// TIA Portal project "Magazyn_v1" (V16)
// Vorlageprojekt für das Buch mit Zielsystem S7-1200

(* hardware
DEVICE "S7-1200-Station_1"  S7-1200 Station
   slot 0: "Baugruppenträger_0"  Rack  V1.0
   slot 1: "PLC_1"  CPU 1211C DC/DC/DC  6ES7 211-1AE40-0XB0  V4.1
DEVICE "HMI_1"  TP900 Comfort SIPLUS
   slot 0: "HMI_1"  TP900 Comfort SIPLUS  6AG1 124-0JC01-4AX0  16.0.0.0
   slot 1: "HMI_RT_1"  TP900 Comfort SIPLUS  6AG1 124-0JC01-4AX0  16.0.0.0
   slot 5: "HMI_1.IE_CP_1"  PROFINET Interface  16.0.0.0
      slot 1: "PROFINET Interface_1"  PROFINET Interface
         slot 1: "Port_1"  Port
         slot 2: "Port_2"  Port
   slot 7: "HMI_1.MPI/DP_CP_1"  MPI/DP Interface  16.0.0.0
*)

// ===== PLC "PLC_1"  CPU 1211C DC/DC/DC =====

VAR_GLOBAL   // PLC tag table "Standard-Variablentabelle"
   "M30.1" AT %M30.1 : Bool;
   "M30.2" AT %M30.2 : Bool;
   "Tag_1" AT %I0.6 : Bool;
   "Tag_2" AT %I0.7 : Bool;
   "Tag_3" AT %Q0.5 : Bool;
   "Tag_4" AT %Q0.6 : Bool;
   "Tag_5" AT %Q0.7 : Bool;
   "box_full" AT %M30.3 : Bool;
   "M1_Conveyor_sec1_1" AT %M30.4 : Bool;
   "M2_Conveyor_sec1_1" AT %M30.5 : Bool;
   "Tag_6" AT %Q1.0 : Bool;
   "M1_Conveyor_sec1_2" AT %M30.6 : Bool;
   "M2_Conveyor_sec1_2" AT %M30.7 : Bool;
   "M1_Conveyor_sec1_3" AT %M31.0 : Bool;
   "M1_Conveyor_sec1_4" AT %M31.2 : Bool;
   "M2_Conveyor_sec1_4" AT %M31.3 : Bool;
   "M1_Conveyor_sec1_5" AT %M31.4 : Bool;
   "M2_Conveyor_sec1_5" AT %M31.5 : Bool;
   "M1_Conveyor_sec1_6" AT %M31.6 : Bool;
   "M2_Conveyor_sec1_6" AT %M31.7 : Bool;
   "M1_Conveyor_sec1_7" AT %M32.0 : Bool;
   "M2_Conveyor_sec1_7" AT %M32.1 : Bool;
   "Tag_7" AT %M32.2 : Bool;
   "pallet_fork_under_box_temp1" AT %M33.0 : Bool;
   "lift_box_temp1" AT %M33.1 : Bool;
   "ready_to_set_up_temp1" AT %M33.2 : Bool;
   "pallet_fork_storage_temp1" AT %M33.3 : Bool;
   "lower_box_temp1" AT %M33.4 : Bool;
   "pallet_fork_storage_withdraw_temp1" AT %M33.5 : Bool;
   "finish_stacker_Crane_sec1" AT %M33.6 : Bool;
   "Tag_8" AT %M33.7 : Bool;
   "is_pallete_elevator" AT %M34.0 : Bool;
   "_move_pallete_temp1" AT %M34.1 : Bool;
   "_move_pallete_temp2" AT %M34.2 : Bool;
   "_move_pallete_temp3" AT %M34.3 : Bool;
   "_move_pallete_temp4" AT %M34.5 : Bool;
   "set_is_pallere" AT %M34.6 : Bool;
   "Tag_9" AT %M34.4 : Bool;
   "pallete_ready_to_load" AT %M34.7 : Bool;
   "palletizing_box" AT %M35.0 : Bool;
   "pop_up_box_M" AT %M35.1 : Bool;
   "pop_up_palletizing_box" AT %M35.2 : Bool;
   "belt_conv_sec2_1_palletizing_box" AT %M35.3 : Bool;
   "belt_conv_sec2_1_palletizing_box_1" AT %M35.4 : Bool;
   "turn_box" AT %MW4 : Int;
   "belt_conv_sec2_1_palletizing_box_2" AT %M35.5 : Bool;
   "parallel_level" AT %M35.6 : Bool;
   "palletizer_finish_level" AT %M35.7 : Bool;
   "pallete_to_storage" AT %M36.0 : Bool;
   "palletizer_elevator_temp1" AT %M36.1 : Bool;
   "pallete_down_temp1" AT %M36.2 : Bool;
   "pallete_to_storage1" AT %M36.3 : Bool;
   "pallete_to_storage3" AT %M36.4 : Bool;
   "pallete_next_load" AT %M36.5 : Bool;
   "pallete_to_storage2" AT %M36.6 : Bool;
   "pallete_to_storage4" AT %M36.7 : Bool;
   "ready_to_set_up_temp1_2" AT %M37.0 : Bool;
   "pallet_fork_under_box_temp1_2" AT %M37.1 : Bool;
   "Tag_10" AT %M37.7 : Bool;
   "Tag_11" AT %M38.0 : Bool;
END_VAR

VAR_GLOBAL   // PLC tag table "Input_Variables_Factory"
   "FactoryIORunning" AT %I0.0 : Bool;
   "FactoryIOPaused" AT %I0.1 : Bool;
   "FactoryIOReset" AT %I0.2 : Bool;
   "Retroreflective Sensor 3 package" AT %I0.3 : Bool;
   "Retroreflective Sensor 4 Weight" AT %I0.4 : Bool;
   "Conveyor Scale 1 Weight (V)" AT %ID30 : Real;
   "M30.0" AT %M30.0 : Bool;
   "Retroreflective Sensor spad" AT %I0.5 : Bool;
   "Conveyor_sec1_1_Retroreflective Sensor" AT %I1.1 : Bool;
   "Conveyor_sec1_2_Retroreflective Sensor" AT %I1.2 : Bool;
   "Conveyor_sec1_3_Retroreflective Sensor" AT %I1.3 : Bool;
   "Conveyor_sec1_4_Retroreflective Sensor" AT %I1.4 : Bool;
   "Conveyor_sec1_5_Retroreflective Sensor" AT %I1.5 : Bool;
   "Conveyor_sec1_6_Retroreflective Sensor" AT %I1.6 : Bool;
   "Conveyor_sec1_7_storage_Retroreflective Sensor" AT %I1.7 : Bool;
   "M2_Conveyor_sec1_3" AT %M31.1 : Bool;
   "Roller_conveyor_sec2_down_1_Retroreflective_Sensor" AT %I2.0 : Bool;
   "Roller_conveyor_sec2_down_2_Retroreflective_Sensor" AT %I2.1 : Bool;
   "Belt_cinv_sec2_1_Retroreflective_Sensor" AT %I2.2 : Bool;
   "Palletizer 2 Elevator (Front Limit)" AT %I2.3 : Bool;
   "Loading_conv_sec2_Retroreflective_Sensor" AT %I2.4 : Bool;
   "Palletizer_Clamped_sensor" AT %I2.5 : Bool;
   "Palletizer_Plate_close" AT %I2.6 : Bool;
   "Palletizer_Pusher_Limit_sensor" AT %I2.7 : Bool;
   "Palletizer 2 Elevator (Back Limit)" AT %I1.0 : Bool;
   "lift_box_temp1_2" AT %M37.2 : Bool;
   "finish_stacker_Crane_sec1_2" AT %M37.3 : Bool;
   "pallet_fork_storage_temp1_2" AT %M37.4 : Bool;
   "lower_box_temp1_2" AT %M37.6 : Bool;
   "pallet_fork_storage_withdraw_temp1_2" AT %M37.5 : Bool;
   "Stacker Crane 2 Moving-X" AT %I3.0 : Bool;
   "Stacker Crane 2 Moving-Z" AT %I3.1 : Bool;
   "paletizer_counter" AT %MW6 : Int;
   "boxes_counter" AT %MW8 : Int;
   "paletizer_number_level" AT %MW16 : Int;
   "boxes_number_package" AT %MW18 : Int;
END_VAR

VAR_GLOBAL   // PLC tag table "Output_Variables_Factory"
   "Belt Conveyor (2m) 1 package" AT %Q0.0 : Bool;
   "Conveyor Scale 1 (+)" AT %Q0.1 : Bool;
   "Pop Up Wheel Sorter 2 (+)" AT %Q0.2 : Bool;
   "Pop Up Wheel Sorter 2 (Right)" AT %Q0.3 : Bool;
   "Belt Conveyor (2m) 7 przed spadem" AT %Q0.4 : Bool;
   "Conveyor_sec1_1" AT %Q1.1 : Bool;
   "Conveyor_sec1_2" AT %Q1.2 : Bool;
   "Conveyor_sec1_3" AT %Q1.3 : Bool;
   "Conveyor_sec1_4" AT %Q1.4 : Bool;
   "Conveyor_sec1_5" AT %Q1.5 : Bool;
   "Conveyor_sec1_6" AT %Q1.6 : Bool;
   "Conveyor_sec1_7_storage" AT %Q1.7 : Bool;
   "Stacker Crane sec1 under_box" AT %Q2.0 : Bool;
   "Stacker Crane sec1 Lift_box" AT %Q2.1 : Bool;
   "Stacker Crane sec1 storage" AT %Q2.2 : Bool;
   "Stacker Crane sec1 Target Position" AT %QD30 : DInt;
   "Belt_cinv_sec2_1" AT %Q2.3 : Bool;
   "Palletizer_belt_forward_sec_2_2" AT %Q2.4 : Bool;
   "Palletizer_turn" AT %Q2.5 : Bool;
   "Palletizer_push" AT %Q2.6 : Bool;
   "Palletizer_clamp" AT %Q2.7 : Bool;
   "Palletizer_open_plate" AT %Q3.0 : Bool;
   "Palletizer_elevator_limit" AT %Q3.1 : Bool;
   "Palletizer_elevator_up" AT %Q3.2 : Bool;
   "Palletizer_elevator_down" AT %Q3.3 : Bool;
   "Palletizer_chain_forward" AT %Q3.4 : Bool;
   "Roller_conveyor_sec2_down_1" AT %Q3.5 : Bool;
   "Roller_conveyor_sec2_down_2" AT %Q3.6 : Bool;
   "Loading_conv_sec2" AT %Q3.7 : Bool;
   "Stacker Crane 2 under_box" AT %Q4.0 : Bool;
   "Stacker Crane 2 Lift_box" AT %Q4.1 : Bool;
   "Stacker Crane 2 storage" AT %Q4.2 : Bool;
   "Stacker Crane 2 Target Position" AT %QD34 : DInt;
END_VAR

VAR_GLOBAL   // PLC tag table "Markers_outputs"
   "_Belt Conveyor (2m) 1 package" AT %M10.0 : Bool;
   "_Conveyor Scale 1 (+)" AT %M10.1 : Bool;
   "_Pop Up Wheel Sorter 2 (+)" AT %M10.2 : Bool;
   "_Pop Up Wheel Sorter 2 (Right)" AT %M10.3 : Bool;
   "_Belt Conveyor (2m) 7 przed spadem" AT %M10.4 : Bool;
   "M10.5" AT %M10.5 : Bool;
   "M10.6" AT %M10.6 : Bool;
   "M10.7" AT %M10.7 : Bool;
   "M11.0" AT %M11.0 : Bool;
   "_Conveyor_sec1_1" AT %M11.1 : Bool;
   "_Conveyor_sec1_2" AT %M11.2 : Bool;
   "_Conveyor_sec1_3" AT %M11.3 : Bool;
   "_Conveyor_sec1_4" AT %M11.4 : Bool;
   "_Conveyor_sec1_5" AT %M11.5 : Bool;
   "_Conveyor_sec1_6" AT %M11.6 : Bool;
   "_Conveyor_sec1_7_storage" AT %M11.7 : Bool;
   "_Stacker Crane sec1 under_box" AT %M12.0 : Bool;
   "_Stacker Crane sec1 Lift_box" AT %M12.1 : Bool;
   "_Stacker Crane sec1 storage" AT %M12.2 : Bool;
   "_Belt_cinv_sec2_1" AT %M12.3 : Bool;
   "_Palletizer_belt_forward_sec_2_2" AT %M12.4 : Bool;
   "_Palletizer_turn" AT %M12.5 : Bool;
   "_Palletizer_push" AT %M12.6 : Bool;
   "_Palletizer_clamp" AT %M12.7 : Bool;
   "_Palletizer_open_plate" AT %M13.0 : Bool;
   "_Palletizer_elevator_limit" AT %M13.1 : Bool;
   "_Palletizer_elevator_up" AT %M13.2 : Bool;
   "_Palletizer_elevator_down" AT %M13.3 : Bool;
   "_Palletizer_chain_forward" AT %M13.4 : Bool;
   "_Roller_conveyor_sec2_down_1" AT %M13.5 : Bool;
   "_Roller_conveyor_sec2_down_2" AT %M13.6 : Bool;
   "_Loading_conv_sec2" AT %M13.7 : Bool;
   "_Stacker Crane 2 under_box" AT %M14.0 : Bool;
   "_Stacker Crane 2 Lift_box" AT %M14.1 : Bool;
   "_Stacker Crane 2 storage" AT %M14.2 : Bool;
   "M14.3" AT %M14.3 : Bool;
   "_Stacker Crane sec1 Target Position" AT %MD20 : DInt;
   "_Stacker Crane sec1 Target Position_temp" AT %MD24 : DInt;
   "_Stacker Crane 2 Target Position" AT %MD38 : DInt;
   "_Stacker Crane 2 Target Position_temp" AT %MD42 : DInt;
END_VAR

VAR_GLOBAL   // PLC tag table "Markers_inputs"
   "_FactoryIORunning" AT %M0.0 : Bool;
   "_FactoryIOPaused" AT %M0.1 : Bool;
   "_FactoryIOReset" AT %M0.2 : Bool;
   "_Retroreflective Sensor 3 package" AT %M0.3 : Bool;
   "_Retroreflective Sensor 4 Weight" AT %M0.4 : Bool;
   "_Retroreflective Sensor spad" AT %M0.5 : Bool;
   "M0.6(1)" AT %M0.6 : Bool;
   "M0.7(1)" AT %M0.7 : Bool;
   "_Palletizer 2 Elevator (Back Limit)" AT %M1.0 : Bool;
   "_Conveyor_sec1_1_Retroreflective Sensor" AT %M1.1 : Bool;
   "_Conveyor_sec1_2_Retroreflective Sensor" AT %M1.2 : Bool;
   "_Conveyor_sec1_3_Retroreflective Sensor" AT %M1.3 : Bool;
   "_Conveyor_sec1_4_Retroreflective Sensor" AT %M1.4 : Bool;
   "_Conveyor_sec1_5_Retroreflective Sensor" AT %M1.5 : Bool;
   "_Conveyor_sec1_6_Retroreflective Sensor" AT %M1.6 : Bool;
   "_Conveyor_sec1_7_storage_Retroreflective Sensor" AT %M1.7 : Bool;
   "_Roller_conveyor_sec2_down_1_Retroreflective_Sensor" AT %M2.0 : Bool;
   "_Roller_conveyor_sec2_down_2_Retroreflective_Sensor" AT %M2.1 : Bool;
   "_Belt_cinv_sec2_1_Retroreflective_Sensor" AT %M2.2 : Bool;
   "_Palletizer 2 Elevator (Front Limit)" AT %M2.3 : Bool;
   "_Loading_conv_sec2_Retroreflective_Sensor" AT %M2.4 : Bool;
   "_Palletizer_Clamped_sensor" AT %M2.5 : Bool;
   "_Palletizer_Plate_close" AT %M2.6 : Bool;
   "_Palletizer_Pusher_Limit_sensor" AT %M2.7 : Bool;
   "_Stacker Crane 2 Moving-X" AT %M3.0 : Bool;
   "_Stacker Crane 2 Moving-Z" AT %M3.1 : Bool;
   "M3.2(1)" AT %M3.2 : Bool;
   "M3.3(1)" AT %M3.3 : Bool;
   "M3.4(1)" AT %M3.4 : Bool;
   "M3.5(1)" AT %M3.5 : Bool;
END_VAR

// folder: System blocks/Program resources

DATA_BLOCK "IEC_Timer_0_DB"   // DB1
{ S7_Optimized_Access := 'TRUE' }
AUTHOR : Simatic
FAMILY : IEC
NAME : IEC_TMR
VERSION : 1.0
// stored: InstanceOfName IEC_TIMER
"IEC_TIMER"
BEGIN
END_DATA_BLOCK

DATA_BLOCK "IEC_Counter_0_DB"   // DB2
{ S7_Optimized_Access := 'TRUE' }
AUTHOR : Simatic
FAMILY : IEC
NAME : CNTR
VERSION : 1.0
// stored: InstanceOfName IEC_COUNTER
"IEC_COUNTER"
BEGIN
END_DATA_BLOCK

DATA_BLOCK "licznik_sekcja_I"   // DB3
{ S7_Optimized_Access := 'TRUE' }
AUTHOR : Simatic
FAMILY : IEC
NAME : CNTR
VERSION : 1.0
// stored: InstanceOfName IEC_COUNTER
"IEC_COUNTER"
BEGIN
END_DATA_BLOCK

DATA_BLOCK "delay_switch_off"   // DB4
{ S7_Optimized_Access := 'TRUE' }
AUTHOR : Simatic
FAMILY : IEC
NAME : IEC_TMR
VERSION : 1.0
// stored: InstanceOfName IEC_TIMER
"IEC_TIMER"
BEGIN
END_DATA_BLOCK

DATA_BLOCK "IEC_Timer_0_DB_1"   // DB5
{ S7_Optimized_Access := 'TRUE' }
AUTHOR : Simatic
FAMILY : IEC
NAME : IEC_TMR
VERSION : 1.0
// stored: InstanceOfName IEC_TIMER
"IEC_TIMER"
BEGIN
END_DATA_BLOCK

DATA_BLOCK "IEC_Timer_0_DB_2"   // DB6
{ S7_Optimized_Access := 'TRUE' }
AUTHOR : Simatic
FAMILY : IEC
NAME : IEC_TMR
VERSION : 1.0
// stored: InstanceOfName IEC_TIMER
"IEC_TIMER"
BEGIN
END_DATA_BLOCK

DATA_BLOCK "IEC_Timer_0_DB_3"   // DB7
{ S7_Optimized_Access := 'TRUE' }
AUTHOR : Simatic
FAMILY : IEC
NAME : IEC_TMR
VERSION : 1.0
// stored: InstanceOfName IEC_TIMER
"IEC_TIMER"
BEGIN
END_DATA_BLOCK

DATA_BLOCK "IEC_Timer_0_DB_4"   // DB8
{ S7_Optimized_Access := 'TRUE' }
AUTHOR : Simatic
FAMILY : IEC
NAME : IEC_TMR
VERSION : 1.0
// stored: InstanceOfName IEC_TIMER
"IEC_TIMER"
BEGIN
END_DATA_BLOCK

DATA_BLOCK "IEC_Timer_0_DB_5"   // DB9
{ S7_Optimized_Access := 'TRUE' }
AUTHOR : Simatic
FAMILY : IEC
NAME : IEC_TMR
VERSION : 1.0
// stored: InstanceOfName IEC_TIMER
"IEC_TIMER"
BEGIN
END_DATA_BLOCK

DATA_BLOCK "IEC_Timer_0_DB_6"   // DB10
{ S7_Optimized_Access := 'TRUE' }
AUTHOR : Simatic
FAMILY : IEC
NAME : IEC_TMR
VERSION : 1.0
// stored: InstanceOfName IEC_TIMER
"IEC_TIMER"
BEGIN
END_DATA_BLOCK

DATA_BLOCK "IEC_Timer_0_DB_7"   // DB11
{ S7_Optimized_Access := 'TRUE' }
AUTHOR : Simatic
FAMILY : IEC
NAME : IEC_TMR
VERSION : 1.0
// stored: InstanceOfName IEC_TIMER
"IEC_TIMER"
BEGIN
END_DATA_BLOCK

DATA_BLOCK "IEC_Timer_0_DB_13"   // DB12
{ S7_Optimized_Access := 'TRUE' }
AUTHOR : Simatic
FAMILY : IEC
NAME : IEC_TMR
VERSION : 1.0
// stored: InstanceOfName IEC_TIMER
"IEC_TIMER"
BEGIN
END_DATA_BLOCK

DATA_BLOCK "IEC_Counter_0_DB_3"   // DB13
{ S7_Optimized_Access := 'TRUE' }
AUTHOR : Simatic
FAMILY : IEC
NAME : CNTR
VERSION : 1.0
// stored: InstanceOfName IEC_COUNTER
"IEC_COUNTER"
BEGIN
END_DATA_BLOCK

DATA_BLOCK "IEC_Timer_0_DB_9"   // DB14
{ S7_Optimized_Access := 'TRUE' }
AUTHOR : Simatic
FAMILY : IEC
NAME : IEC_TMR
VERSION : 1.0
// stored: InstanceOfName IEC_TIMER
"IEC_TIMER"
BEGIN
END_DATA_BLOCK

DATA_BLOCK "IEC_Timer_0_DB_10"   // DB15
{ S7_Optimized_Access := 'TRUE' }
AUTHOR : Simatic
FAMILY : IEC
NAME : IEC_TMR
VERSION : 1.0
// stored: InstanceOfName IEC_TIMER
"IEC_TIMER"
BEGIN
END_DATA_BLOCK

DATA_BLOCK "IEC_Counter_0_DB_4"   // DB16
{ S7_Optimized_Access := 'TRUE' }
AUTHOR : Simatic
FAMILY : IEC
NAME : CNTR
VERSION : 1.0
// stored: InstanceOfName IEC_COUNTER
"IEC_COUNTER"
BEGIN
END_DATA_BLOCK

DATA_BLOCK "IEC_Timer_0_DB_14"   // DB18
{ S7_Optimized_Access := 'TRUE' }
AUTHOR : Simatic
FAMILY : IEC
NAME : IEC_TMR
VERSION : 1.0
// stored: InstanceOfName IEC_TIMER
"IEC_TIMER"
BEGIN
END_DATA_BLOCK

DATA_BLOCK "IEC_Timer_0_DB_15"   // DB19
{ S7_Optimized_Access := 'TRUE' }
AUTHOR : Simatic
FAMILY : IEC
NAME : IEC_TMR
VERSION : 1.0
// stored: InstanceOfName IEC_TIMER
"IEC_TIMER"
BEGIN
END_DATA_BLOCK

DATA_BLOCK "IEC_Timer_0_DB_16"   // DB20
{ S7_Optimized_Access := 'TRUE' }
AUTHOR : Simatic
FAMILY : IEC
NAME : IEC_TMR
VERSION : 1.0
// stored: InstanceOfName IEC_TIMER
"IEC_TIMER"
BEGIN
END_DATA_BLOCK

DATA_BLOCK "IEC_Timer_0_DB_17"   // DB21
{ S7_Optimized_Access := 'TRUE' }
AUTHOR : Simatic
FAMILY : IEC
NAME : IEC_TMR
VERSION : 1.0
// stored: InstanceOfName IEC_TIMER
"IEC_TIMER"
BEGIN
END_DATA_BLOCK

DATA_BLOCK "licznik_sekcja_II"   // DB22
{ S7_Optimized_Access := 'TRUE' }
AUTHOR : Simatic
FAMILY : IEC
NAME : CNTR
VERSION : 1.0
// stored: InstanceOfName IEC_COUNTER
"IEC_COUNTER"
BEGIN
END_DATA_BLOCK

DATA_BLOCK "IEC_Timer_0_DB_19"   // DB23
{ S7_Optimized_Access := 'TRUE' }
AUTHOR : Simatic
FAMILY : IEC
NAME : IEC_TMR
VERSION : 1.0
// stored: InstanceOfName IEC_TIMER
"IEC_TIMER"
BEGIN
END_DATA_BLOCK

DATA_BLOCK "licznik_sekcja_II_two_levels"   // DB24
{ S7_Optimized_Access := 'TRUE' }
AUTHOR : Simatic
FAMILY : IEC
NAME : CNTR
VERSION : 1.0
// stored: InstanceOfName IEC_COUNTER
"IEC_COUNTER"
BEGIN
END_DATA_BLOCK

DATA_BLOCK "IEC_Timer_0_DB_20"   // DB25
{ S7_Optimized_Access := 'TRUE' }
AUTHOR : Simatic
FAMILY : IEC
NAME : IEC_TMR
VERSION : 1.0
// stored: InstanceOfName IEC_TIMER
"IEC_TIMER"
BEGIN
END_DATA_BLOCK

DATA_BLOCK "IEC_Timer_0_DB_18"   // DB26
{ S7_Optimized_Access := 'TRUE' }
AUTHOR : Simatic
FAMILY : IEC
NAME : IEC_TMR
VERSION : 1.0
// stored: InstanceOfName IEC_TIMER
"IEC_TIMER"
BEGIN
END_DATA_BLOCK

DATA_BLOCK "IEC_Timer_0_DB_21"   // DB27
{ S7_Optimized_Access := 'TRUE' }
AUTHOR : Simatic
FAMILY : IEC
NAME : IEC_TMR
VERSION : 1.0
// stored: InstanceOfName IEC_TIMER
"IEC_TIMER"
BEGIN
END_DATA_BLOCK

DATA_BLOCK "IEC_Counter_0_DB_1"   // DB28
{ S7_Optimized_Access := 'TRUE' }
AUTHOR : Simatic
FAMILY : IEC
NAME : CNTR
VERSION : 1.0
// stored: InstanceOfName IEC_COUNTER
"IEC_COUNTER"
BEGIN
END_DATA_BLOCK

DATA_BLOCK "IEC_Timer_0_DB_22"   // DB29
{ S7_Optimized_Access := 'TRUE' }
AUTHOR : Simatic
FAMILY : IEC
NAME : IEC_TMR
VERSION : 1.0
// stored: InstanceOfName IEC_TIMER
"IEC_TIMER"
BEGIN
END_DATA_BLOCK

DATA_BLOCK "IEC_Timer_0_DB_23"   // DB30
{ S7_Optimized_Access := 'TRUE' }
AUTHOR : Simatic
FAMILY : IEC
NAME : IEC_TMR
VERSION : 1.0
// stored: InstanceOfName IEC_TIMER
"IEC_TIMER"
BEGIN
END_DATA_BLOCK

DATA_BLOCK "IEC_Timer_0_DB_24"   // DB31
{ S7_Optimized_Access := 'TRUE' }
AUTHOR : Simatic
FAMILY : IEC
NAME : IEC_TMR
VERSION : 1.0
// stored: InstanceOfName IEC_TIMER
"IEC_TIMER"
BEGIN
END_DATA_BLOCK

DATA_BLOCK "IEC_Timer_0_DB_25"   // DB32
{ S7_Optimized_Access := 'TRUE' }
AUTHOR : Simatic
FAMILY : IEC
NAME : IEC_TMR
VERSION : 1.0
// stored: InstanceOfName IEC_TIMER
"IEC_TIMER"
BEGIN
END_DATA_BLOCK

DATA_BLOCK "IEC_Counter_0_DB_2"   // DB33
{ S7_Optimized_Access := 'TRUE' }
AUTHOR : Simatic
FAMILY : IEC
NAME : CNTR
VERSION : 1.0
// stored: InstanceOfName IEC_COUNTER
"IEC_COUNTER"
BEGIN
END_DATA_BLOCK

DATA_BLOCK "IEC_Timer_0_DB_26"   // DB34
{ S7_Optimized_Access := 'TRUE' }
AUTHOR : Simatic
FAMILY : IEC
NAME : IEC_TMR
VERSION : 1.0
// stored: InstanceOfName IEC_TIMER
"IEC_TIMER"
BEGIN
END_DATA_BLOCK

DATA_BLOCK "IEC_Timer_0_DB_27"   // DB35
{ S7_Optimized_Access := 'TRUE' }
AUTHOR : Simatic
FAMILY : IEC
NAME : IEC_TMR
VERSION : 1.0
// stored: InstanceOfName IEC_TIMER
"IEC_TIMER"
BEGIN
END_DATA_BLOCK

DATA_BLOCK "IEC_Timer_0_DB_28"   // DB36
{ S7_Optimized_Access := 'TRUE' }
AUTHOR : Simatic
FAMILY : IEC
NAME : IEC_TMR
VERSION : 1.0
// stored: InstanceOfName IEC_TIMER
"IEC_TIMER"
BEGIN
END_DATA_BLOCK

DATA_BLOCK "IEC_Timer_0_DB_29"   // DB37
{ S7_Optimized_Access := 'TRUE' }
AUTHOR : Simatic
FAMILY : IEC
NAME : IEC_TMR
VERSION : 1.0
// stored: InstanceOfName IEC_TIMER
"IEC_TIMER"
BEGIN
END_DATA_BLOCK

DATA_BLOCK "IEC_Timer_0_DB_30"   // DB38
{ S7_Optimized_Access := 'TRUE' }
AUTHOR : Simatic
FAMILY : IEC
NAME : IEC_TMR
VERSION : 1.0
// stored: InstanceOfName IEC_TIMER
"IEC_TIMER"
BEGIN
END_DATA_BLOCK

DATA_BLOCK "IEC_Timer_0_DB_31"   // DB39
{ S7_Optimized_Access := 'TRUE' }
AUTHOR : Simatic
FAMILY : IEC
NAME : IEC_TMR
VERSION : 1.0
// stored: InstanceOfName IEC_TIMER
"IEC_TIMER"
BEGIN
END_DATA_BLOCK

DATA_BLOCK "IEC_Timer_0_DB_32"   // DB40
{ S7_Optimized_Access := 'TRUE' }
AUTHOR : Simatic
FAMILY : IEC
NAME : IEC_TMR
VERSION : 1.0
// stored: InstanceOfName IEC_TIMER
"IEC_TIMER"
BEGIN
END_DATA_BLOCK

DATA_BLOCK "IEC_Timer_0_DB_33"   // DB41
{ S7_Optimized_Access := 'TRUE' }
AUTHOR : Simatic
FAMILY : IEC
NAME : IEC_TMR
VERSION : 1.0
// stored: InstanceOfName IEC_TIMER
"IEC_TIMER"
BEGIN
END_DATA_BLOCK

DATA_BLOCK "IEC_Timer_0_DB_34"   // DB42
{ S7_Optimized_Access := 'TRUE' }
AUTHOR : Simatic
FAMILY : IEC
NAME : IEC_TMR
VERSION : 1.0
// stored: InstanceOfName IEC_TIMER
"IEC_TIMER"
BEGIN
END_DATA_BLOCK

DATA_BLOCK "IEC_Timer_0_DB_35"   // DB43
{ S7_Optimized_Access := 'TRUE' }
AUTHOR : Simatic
FAMILY : IEC
NAME : IEC_TMR
VERSION : 1.0
// stored: InstanceOfName IEC_TIMER
"IEC_TIMER"
BEGIN
END_DATA_BLOCK

DATA_BLOCK "IEC_Timer_0_DB_36"   // DB44
{ S7_Optimized_Access := 'TRUE' }
AUTHOR : Simatic
FAMILY : IEC
NAME : IEC_TMR
VERSION : 1.0
// stored: InstanceOfName IEC_TIMER
"IEC_TIMER"
BEGIN
END_DATA_BLOCK

DATA_BLOCK "IEC_Timer_0_DB_37"   // DB45
{ S7_Optimized_Access := 'TRUE' }
AUTHOR : Simatic
FAMILY : IEC
NAME : IEC_TMR
VERSION : 1.0
// stored: InstanceOfName IEC_TIMER
"IEC_TIMER"
BEGIN
END_DATA_BLOCK

DATA_BLOCK "IEC_Timer_0_DB_38"   // DB46
{ S7_Optimized_Access := 'TRUE' }
AUTHOR : Simatic
FAMILY : IEC
NAME : IEC_TMR
VERSION : 1.0
// stored: InstanceOfName IEC_TIMER
"IEC_TIMER"
BEGIN
END_DATA_BLOCK

// folder: (top level)

FUNCTION "stacker_crane_2" : Void   // FC1, LAD
{ S7_Optimized_Access := 'TRUE' }
VERSION : 0.1
   VAR_TEMP
      mem5 : Bool;
      mem6 : Bool;
      mem7 : Bool;
   END_VAR
   VAR_TEMP   // added for the SCL form of the ladder/FBD networks
      _w1 : Bool;
      _w2 : Bool;
   END_VAR
BEGIN

REGION Network 2: Section1_pallete_fork
   // podjazd pod palete
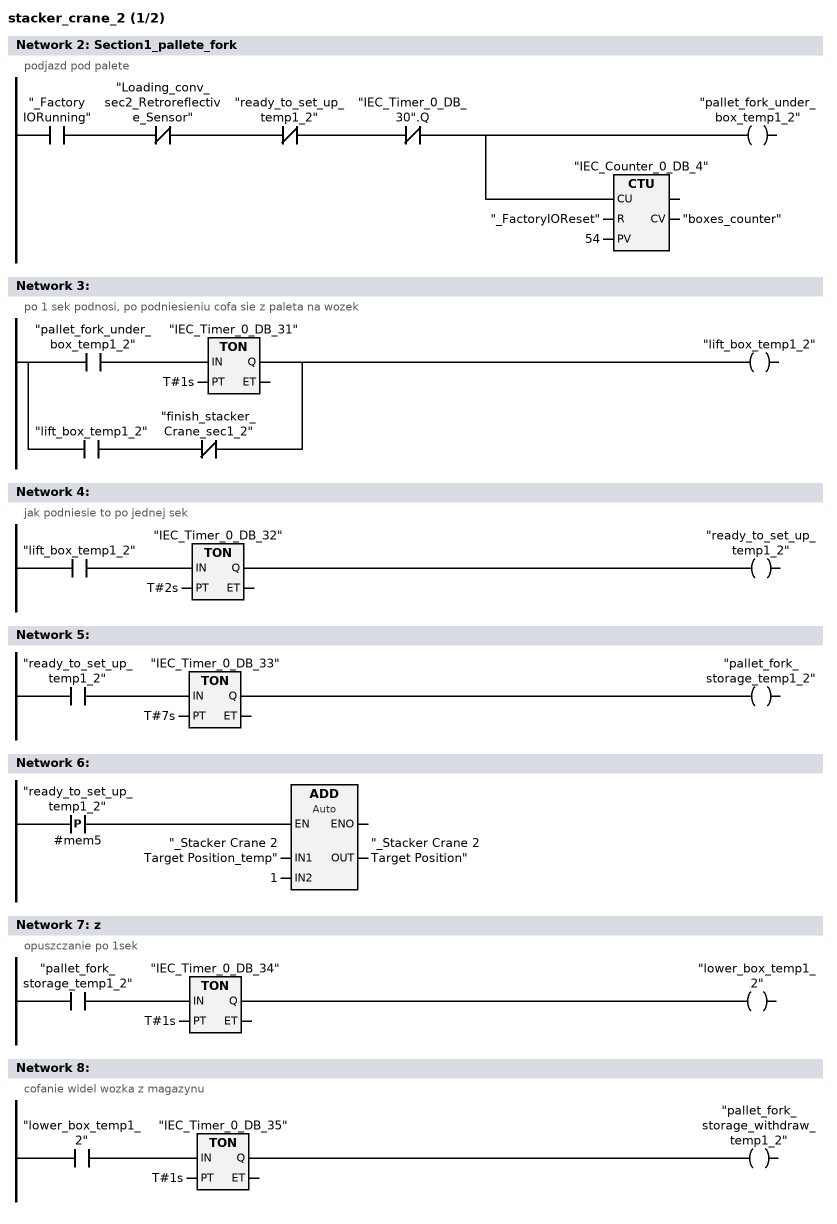
   "pallet_fork_under_box_temp1_2" := "_FactoryIORunning" AND NOT "Loading_conv_sec2_Retroreflective_Sensor" AND NOT "ready_to_set_up_temp1_2" AND NOT "IEC_Timer_0_DB_30".Q;
   "IEC_Counter_0_DB_4".CTU(CU := "pallet_fork_under_box_temp1_2",
                           R := "_FactoryIOReset",
                           PV := 54,
                           CV => "boxes_counter");
END_REGION

REGION Network 3
   // po 1 sek podnosi, po podniesieniu cofa sie z paleta na wozek
   "IEC_Timer_0_DB_31".TON(IN := "pallet_fork_under_box_temp1_2", PT := T#1s);
   "lift_box_temp1_2" := "IEC_Timer_0_DB_31".Q OR ("lift_box_temp1_2" AND NOT "finish_stacker_Crane_sec1_2");
END_REGION

REGION Network 4
   // jak podniesie to po jednej sek
   "IEC_Timer_0_DB_32".TON(IN := "lift_box_temp1_2", PT := T#2s);
   "ready_to_set_up_temp1_2" := "IEC_Timer_0_DB_32".Q;
END_REGION

REGION Network 5
   "IEC_Timer_0_DB_33".TON(IN := "ready_to_set_up_temp1_2", PT := T#7s);
   "pallet_fork_storage_temp1_2" := "IEC_Timer_0_DB_33".Q;
END_REGION

REGION Network 6
   RUNG wire#powerrail
      P_Contact(operand := "ready_to_set_up_temp1_2", bit := #mem5)
      Add(in1 := "_Stacker Crane 2 Target Position_temp", in2 := 1, out => "_Stacker Crane 2 Target Position")
   END_RUNG
   // the same network as SCL:
   #_w1 := "ready_to_set_up_temp1_2" AND NOT #mem5;   // rising edge of "ready_to_set_up_temp1_2"
   #mem5 := "ready_to_set_up_temp1_2";
   IF #_w1 THEN "_Stacker Crane 2 Target Position" := "_Stacker Crane 2 Target Position_temp" + 1; END_IF;
END_REGION

REGION Network 7: z
   // opuszczanie po 1sek
   "IEC_Timer_0_DB_34".TON(IN := "pallet_fork_storage_temp1_2", PT := T#1s);
   "lower_box_temp1_2" := "IEC_Timer_0_DB_34".Q;
END_REGION

REGION Network 8
   // cofanie widel wozka z magazynu
   "IEC_Timer_0_DB_35".TON(IN := "lower_box_temp1_2", PT := T#1s);
   "pallet_fork_storage_withdraw_temp1_2" := "IEC_Timer_0_DB_35".Q;
END_REGION

REGION Network 9
   // powrot na pozycje startowa widlaka
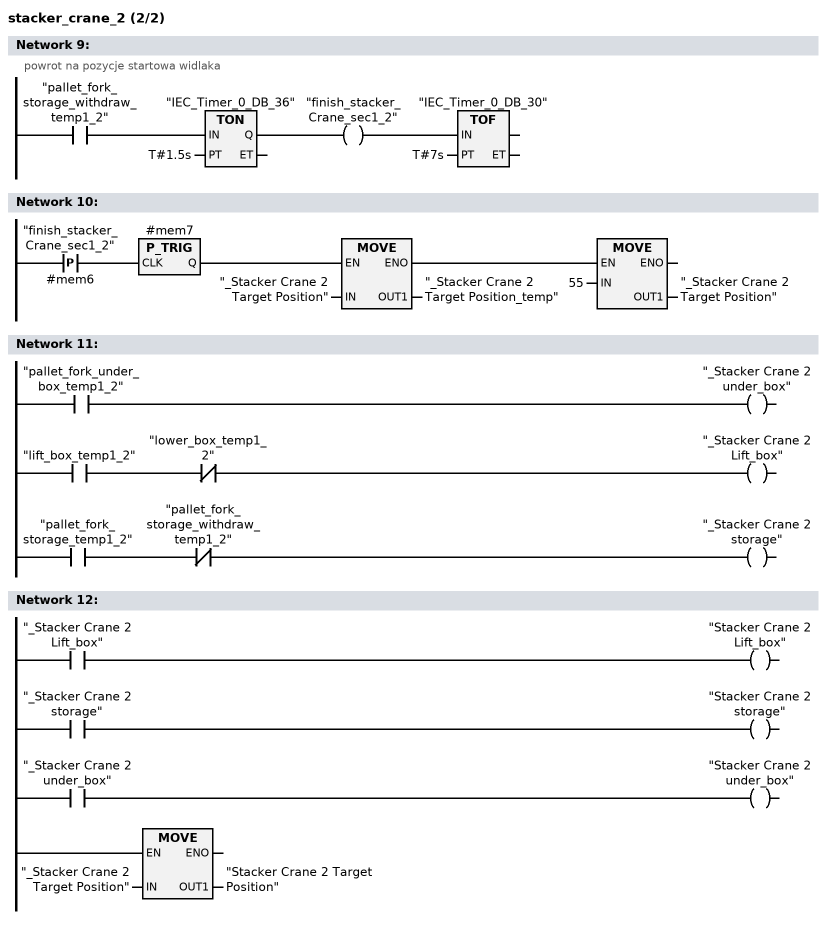
   "IEC_Timer_0_DB_36".TON(IN := "pallet_fork_storage_withdraw_temp1_2", PT := T#1.5s);
   "finish_stacker_Crane_sec1_2" := "IEC_Timer_0_DB_36".Q;
   "IEC_Timer_0_DB_30".TOF(IN := "IEC_Timer_0_DB_36".Q, PT := T#7s);
END_REGION

REGION Network 10
   RUNG wire#powerrail
      P_Contact(operand := "finish_stacker_Crane_sec1_2", bit := #mem6)
      P_Trig( #mem7 )
      Move(in := "_Stacker Crane 2 Target Position", out1 => "_Stacker Crane 2 Target Position_temp")
      Move(in := 55, out1 => "_Stacker Crane 2 Target Position")
   END_RUNG
   // the same network as SCL:
   #_w1 := "finish_stacker_Crane_sec1_2" AND NOT #mem6;   // rising edge of "finish_stacker_Crane_sec1_2"
   #mem6 := "finish_stacker_Crane_sec1_2";
   #_w2 := #_w1 AND NOT #mem7;   // rising edge
   #mem7 := #_w1;
   IF #_w2 THEN
       "_Stacker Crane 2 Target Position_temp" := "_Stacker Crane 2 Target Position";
       "_Stacker Crane 2 Target Position" := 55;
   END_IF;
END_REGION

REGION Network 11
   RUNG wire#powerrail
      Contact( "pallet_fork_under_box_temp1_2" )
      Coil( "_Stacker Crane 2 under_box" )
   END_RUNG
   RUNG wire#powerrail
      Contact( "lift_box_temp1_2" )
      I_Contact( "lower_box_temp1_2" )
      Coil( "_Stacker Crane 2 Lift_box" )
   END_RUNG
   RUNG wire#powerrail
      Contact( "pallet_fork_storage_temp1_2" )
      I_Contact( "pallet_fork_storage_withdraw_temp1_2" )
      Coil( "_Stacker Crane 2 storage" )
   END_RUNG
   // the same network as SCL:
   "_Stacker Crane 2 under_box" := "pallet_fork_under_box_temp1_2";
   "_Stacker Crane 2 Lift_box" := "lift_box_temp1_2" AND NOT "lower_box_temp1_2";
   "_Stacker Crane 2 storage" := "pallet_fork_storage_temp1_2" AND NOT "pallet_fork_storage_withdraw_temp1_2";
END_REGION

REGION Network 12
   RUNG wire#powerrail
      Contact( "_Stacker Crane 2 Lift_box" )
      Coil( "Stacker Crane 2 Lift_box" )
   END_RUNG
   RUNG wire#powerrail
      Contact( "_Stacker Crane 2 storage" )
      Coil( "Stacker Crane 2 storage" )
   END_RUNG
   RUNG wire#powerrail
      Contact( "_Stacker Crane 2 under_box" )
      Coil( "Stacker Crane 2 under_box" )
   END_RUNG
   RUNG wire#powerrail
      Move(in := "_Stacker Crane 2 Target Position", out1 => "Stacker Crane 2 Target Position")
   END_RUNG
   // the same network as SCL:
   "Stacker Crane 2 Lift_box" := "_Stacker Crane 2 Lift_box";
   "Stacker Crane 2 storage" := "_Stacker Crane 2 storage";
   "Stacker Crane 2 under_box" := "_Stacker Crane 2 under_box";
   "Stacker Crane 2 Target Position" := "_Stacker Crane 2 Target Position";
END_REGION
END_FUNCTION

FUNCTION "MHJ-PLC-Lab-Function-S71200" : Void   // FC9000, SCL
{ S7_Optimized_Access := 'TRUE' }
VERSION : 0.1
   VAR_TEMP
      rdTimeReturn : Int;
      outputTime : DTL;
      SyncVal : Byte;
      forVal : Int;
      forVal_2 : Int;
      Value : Byte;
   END_VAR
   VAR CONSTANT
      CompVal : Byte := 16#34;
      Value_01 : Byte := 16#11;
      Value_01_DW : DWord := 16#A165_D992;
      Value_02_DW : DWord := 16#58BE_4401;
   END_VAR
BEGIN

   #Value:=PEEK(area := 16#82,
        dbNumber := 0,
        byteOffset := 511);
   #Value := #Value + 1;

   POKE(area := 16#82,
        dbNumber := 0,
        byteOffset := 511,
        value := #Value);

   POKE(area:=16#81,
        dbNumber:=0,
        byteOffset:=1016,
        value:=#Value_01_DW);
   POKE(area := 16#81,
        dbNumber := 0,
        byteOffset := 1020,
        value := #Value_02_DW);

   POKE(area := 16#81,
        dbNumber := 0,
        byteOffset := 511,
        value := B#16#00);

   FOR #forVal := 0 TO 120 DO
       FOR #forVal_2:=0 TO 10 DO
           #rdTimeReturn:=RD_SYS_T(#outputTime);
           #rdTimeReturn := WR_SYS_T(#outputTime);
           #rdTimeReturn := RD_SYS_T(#outputTime);
           #rdTimeReturn := WR_SYS_T(#outputTime);
       END_FOR;
       #SyncVal:= PEEK(area := 16#81,
                      dbNumber := 0,
                      byteOffset := 511);
       IF #SyncVal = #CompVal THEN
          GOTO M_1;
       END_IF;
   END_FOR;
   RETURN;

   M_1:
   POKE(area := 16#81,
        dbNumber := 0,
        byteOffset := 511,
        value := B#16#0);
END_FUNCTION

ORGANIZATION_BLOCK "Main"   // OB1, LAD, ProgramCycle
TITLE = "Main Program Sweep (Cycle)"
{ S7_Optimized_Access := 'TRUE' }
VERSION : 0.1
   VAR_INPUT
      Initial_Call : Bool;   // Initial call of this OB
      Remanence : Bool;   // =True, if remanent data are available
   END_VAR
   VAR_TEMP
      mem1 : Bool;
      mem2 : Bool;
      mem3 : Bool;
      _box_full : Bool;
      M1_Conveyor_sec1_1 : Bool;
      M2_Conveyor_sec1_1 : Bool;
      mem4 : Bool;
      mem5 : Bool;
      mem6 : Bool;
      mem7 : Bool;
      mem8 : Bool;
      sr1 : Bool;
      sr2 : Bool;
      mem9 : Bool;
      mem10 : Bool;
      mem11 : Bool;
      mem12 : Bool;
      mem13 : Bool;
      mem14 : Bool;
      mem15 : Bool;
      mem16 : Bool;
      mem17 : Bool;
      mem18 : Bool;
      mem19 : Bool;
      mem20 : Bool;
   END_VAR
   VAR_TEMP   // added for the SCL form of the ladder/FBD networks
      _w1 : Bool;
      _w2 : Bool;
   END_VAR
BEGIN

REGION Network 1: Konnektierungsbaustein für PLC-Lab
   // Im Netzwerk 1 wird der Konnektierungsbaustein für PLC-Lab aufgerufen.
   // Dieser Aufruf darf nicht entfernt werden!
   // Enable connention with Factory I/O
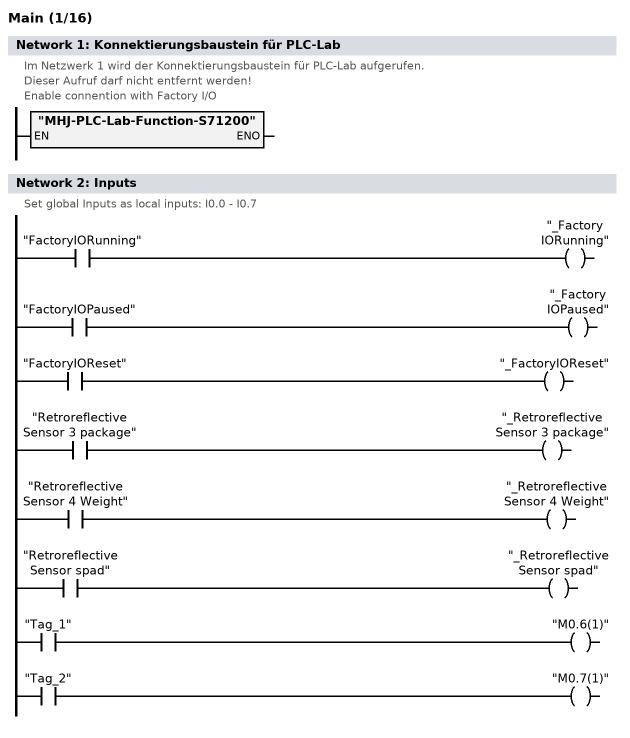
   RUNG wire#powerrail
      "MHJ-PLC-Lab-Function-S71200"()
   END_RUNG
   // the same network as SCL:
   "MHJ-PLC-Lab-Function-S71200"();
END_REGION

REGION Network 2: Inputs
   // Set global Inputs as local inputs: I0.0 - I0.7
   RUNG wire#powerrail
      Contact( "FactoryIORunning" )
      Coil( "_FactoryIORunning" )
   END_RUNG
   RUNG wire#powerrail
      Contact( "FactoryIOPaused" )
      Coil( "_FactoryIOPaused" )
   END_RUNG
   RUNG wire#powerrail
      Contact( "FactoryIOReset" )
      Coil( "_FactoryIOReset" )
   END_RUNG
   RUNG wire#powerrail
      Contact( "Retroreflective Sensor 3 package" )
      Coil( "_Retroreflective Sensor 3 package" )
   END_RUNG
   RUNG wire#powerrail
      Contact( "Retroreflective Sensor 4 Weight" )
      Coil( "_Retroreflective Sensor 4 Weight" )
   END_RUNG
   RUNG wire#powerrail
      Contact( "Retroreflective Sensor spad" )
      Coil( "_Retroreflective Sensor spad" )
   END_RUNG
   RUNG wire#powerrail
      Contact( "Tag_1" )
      Coil( "M0.6(1)" )
   END_RUNG
   RUNG wire#powerrail
      Contact( "Tag_2" )
      Coil( "M0.7(1)" )
   END_RUNG
   // the same network as SCL:
   "_FactoryIORunning" := "FactoryIORunning";
   "_FactoryIOPaused" := "FactoryIOPaused";
   "_FactoryIOReset" := "FactoryIOReset";
   "_Retroreflective Sensor 3 package" := "Retroreflective Sensor 3 package";
   "_Retroreflective Sensor 4 Weight" := "Retroreflective Sensor 4 Weight";
   "_Retroreflective Sensor spad" := "Retroreflective Sensor spad";
   "M0.6(1)" := "Tag_1";
   "M0.7(1)" := "Tag_2";
END_REGION

REGION Network 3
   // Set global Inputs as local inputs: I1.0 - I1.7
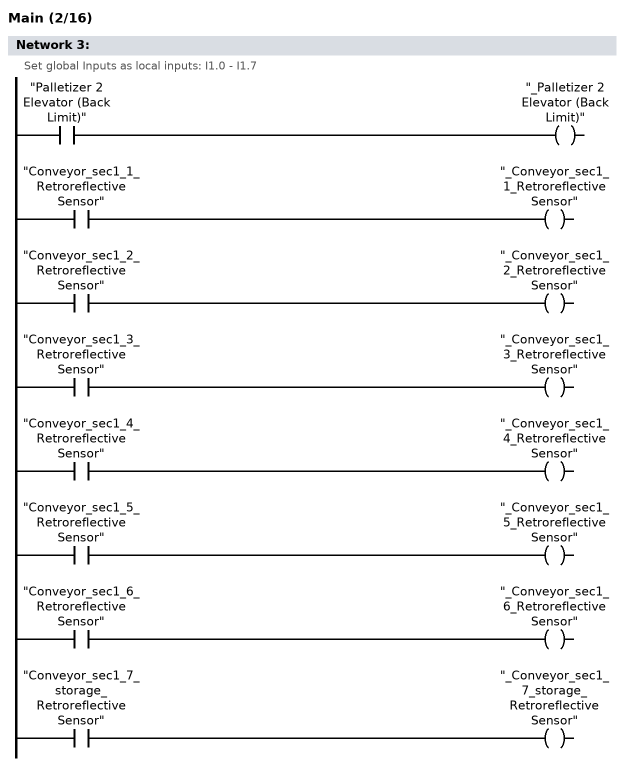
   RUNG wire#powerrail
      Contact( "Palletizer 2 Elevator (Back Limit)" )
      Coil( "_Palletizer 2 Elevator (Back Limit)" )
   END_RUNG
   RUNG wire#powerrail
      Contact( "Conveyor_sec1_1_Retroreflective Sensor" )
      Coil( "_Conveyor_sec1_1_Retroreflective Sensor" )
   END_RUNG
   RUNG wire#powerrail
      Contact( "Conveyor_sec1_2_Retroreflective Sensor" )
      Coil( "_Conveyor_sec1_2_Retroreflective Sensor" )
   END_RUNG
   RUNG wire#powerrail
      Contact( "Conveyor_sec1_3_Retroreflective Sensor" )
      Coil( "_Conveyor_sec1_3_Retroreflective Sensor" )
   END_RUNG
   RUNG wire#powerrail
      Contact( "Conveyor_sec1_4_Retroreflective Sensor" )
      Coil( "_Conveyor_sec1_4_Retroreflective Sensor" )
   END_RUNG
   RUNG wire#powerrail
      Contact( "Conveyor_sec1_5_Retroreflective Sensor" )
      Coil( "_Conveyor_sec1_5_Retroreflective Sensor" )
   END_RUNG
   RUNG wire#powerrail
      Contact( "Conveyor_sec1_6_Retroreflective Sensor" )
      Coil( "_Conveyor_sec1_6_Retroreflective Sensor" )
   END_RUNG
   RUNG wire#powerrail
      Contact( "Conveyor_sec1_7_storage_Retroreflective Sensor" )
      Coil( "_Conveyor_sec1_7_storage_Retroreflective Sensor" )
   END_RUNG
   // the same network as SCL:
   "_Palletizer 2 Elevator (Back Limit)" := "Palletizer 2 Elevator (Back Limit)";
   "_Conveyor_sec1_1_Retroreflective Sensor" := "Conveyor_sec1_1_Retroreflective Sensor";
   "_Conveyor_sec1_2_Retroreflective Sensor" := "Conveyor_sec1_2_Retroreflective Sensor";
   "_Conveyor_sec1_3_Retroreflective Sensor" := "Conveyor_sec1_3_Retroreflective Sensor";
   "_Conveyor_sec1_4_Retroreflective Sensor" := "Conveyor_sec1_4_Retroreflective Sensor";
   "_Conveyor_sec1_5_Retroreflective Sensor" := "Conveyor_sec1_5_Retroreflective Sensor";
   "_Conveyor_sec1_6_Retroreflective Sensor" := "Conveyor_sec1_6_Retroreflective Sensor";
   "_Conveyor_sec1_7_storage_Retroreflective Sensor" := "Conveyor_sec1_7_storage_Retroreflective Sensor";
END_REGION

REGION Network 4
   // Set global Inputs as local inputs: I2.0 - I2.7
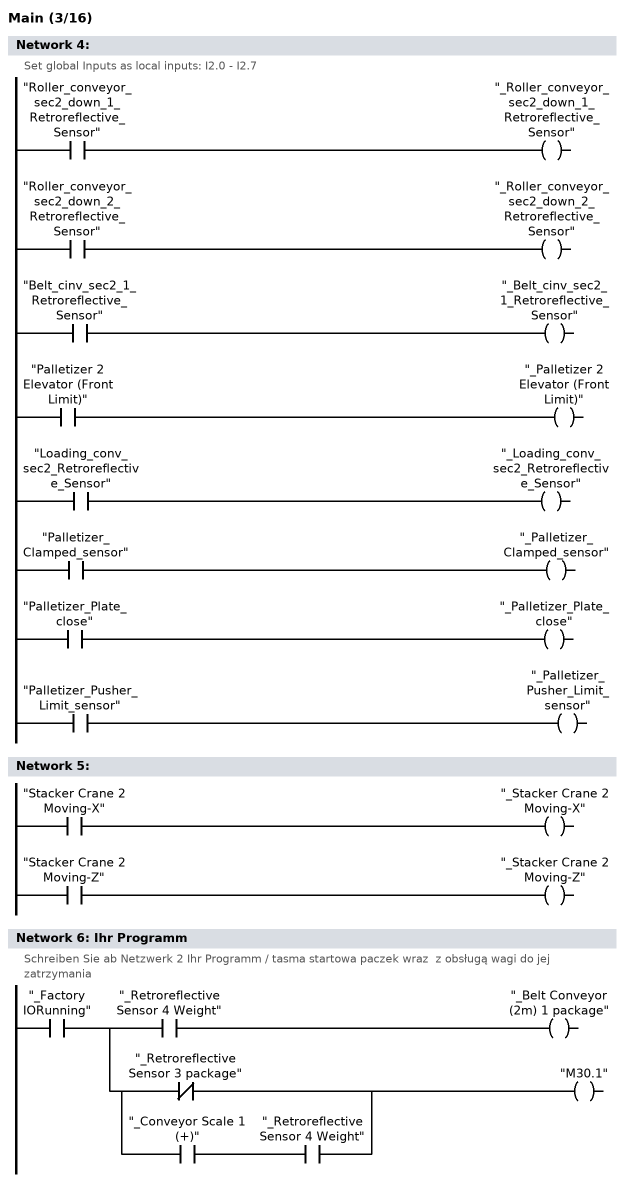
   RUNG wire#powerrail
      Contact( "Roller_conveyor_sec2_down_1_Retroreflective_Sensor" )
      Coil( "_Roller_conveyor_sec2_down_1_Retroreflective_Sensor" )
   END_RUNG
   RUNG wire#powerrail
      Contact( "Roller_conveyor_sec2_down_2_Retroreflective_Sensor" )
      Coil( "_Roller_conveyor_sec2_down_2_Retroreflective_Sensor" )
   END_RUNG
   RUNG wire#powerrail
      Contact( "Belt_cinv_sec2_1_Retroreflective_Sensor" )
      Coil( "_Belt_cinv_sec2_1_Retroreflective_Sensor" )
   END_RUNG
   RUNG wire#powerrail
      Contact( "Palletizer 2 Elevator (Front Limit)" )
      Coil( "_Palletizer 2 Elevator (Front Limit)" )
   END_RUNG
   RUNG wire#powerrail
      Contact( "Loading_conv_sec2_Retroreflective_Sensor" )
      Coil( "_Loading_conv_sec2_Retroreflective_Sensor" )
   END_RUNG
   RUNG wire#powerrail
      Contact( "Palletizer_Clamped_sensor" )
      Coil( "_Palletizer_Clamped_sensor" )
   END_RUNG
   RUNG wire#powerrail
      Contact( "Palletizer_Plate_close" )
      Coil( "_Palletizer_Plate_close" )
   END_RUNG
   RUNG wire#powerrail
      Contact( "Palletizer_Pusher_Limit_sensor" )
      Coil( "_Palletizer_Pusher_Limit_sensor" )
   END_RUNG
   // the same network as SCL:
   "_Roller_conveyor_sec2_down_1_Retroreflective_Sensor" := "Roller_conveyor_sec2_down_1_Retroreflective_Sensor";
   "_Roller_conveyor_sec2_down_2_Retroreflective_Sensor" := "Roller_conveyor_sec2_down_2_Retroreflective_Sensor";
   "_Belt_cinv_sec2_1_Retroreflective_Sensor" := "Belt_cinv_sec2_1_Retroreflective_Sensor";
   "_Palletizer 2 Elevator (Front Limit)" := "Palletizer 2 Elevator (Front Limit)";
   "_Loading_conv_sec2_Retroreflective_Sensor" := "Loading_conv_sec2_Retroreflective_Sensor";
   "_Palletizer_Clamped_sensor" := "Palletizer_Clamped_sensor";
   "_Palletizer_Plate_close" := "Palletizer_Plate_close";
   "_Palletizer_Pusher_Limit_sensor" := "Palletizer_Pusher_Limit_sensor";
END_REGION

REGION Network 5
   RUNG wire#powerrail
      Contact( "Stacker Crane 2 Moving-X" )
      Coil( "_Stacker Crane 2 Moving-X" )
   END_RUNG
   RUNG wire#powerrail
      Contact( "Stacker Crane 2 Moving-Z" )
      Coil( "_Stacker Crane 2 Moving-Z" )
   END_RUNG
   // the same network as SCL:
   "_Stacker Crane 2 Moving-X" := "Stacker Crane 2 Moving-X";
   "_Stacker Crane 2 Moving-Z" := "Stacker Crane 2 Moving-Z";
END_REGION

REGION Network 6: Ihr Programm
   // Schreiben Sie ab Netzwerk 2 Ihr Programm / tasma startowa paczek wraz  z obsługą wagi do jej zatrzymania
   RUNG wire#powerrail
      Contact( "_FactoryIORunning" )
      wire#w1
      Contact( "_Retroreflective Sensor 4 Weight" )
      Coil( "_Belt Conveyor (2m) 1 package" )
   END_RUNG
   RUNG wire#w1
      I_Contact( "_Retroreflective Sensor 3 package" )
      wire#w2
      Coil( "M30.1" )
   END_RUNG
   RUNG wire#w1
      Contact( "_Conveyor Scale 1 (+)" )
      Contact( "_Retroreflective Sensor 4 Weight" )
   END_RUNG wire#w2
   // the same network as SCL:
   "_Belt Conveyor (2m) 1 package" := "_FactoryIORunning" AND "_Retroreflective Sensor 4 Weight";
   "M30.1" := "_FactoryIORunning" AND (NOT "_Retroreflective Sensor 3 package" OR ("_Conveyor Scale 1 (+)" AND "_Retroreflective Sensor 4 Weight"));
END_REGION

REGION Network 7
   // rolki dla paczki M oraz zalaczenie tasmy - warunki
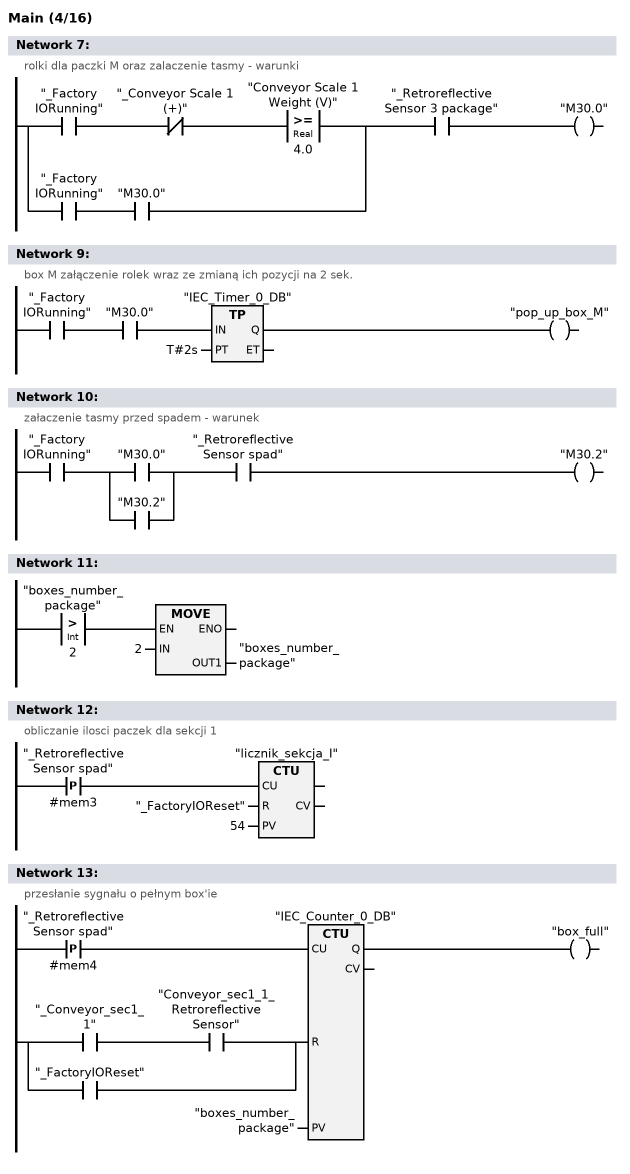
   RUNG wire#powerrail
      Contact( "_FactoryIORunning" )
      I_Contact( "_Conveyor Scale 1 (+)" )
      { S7_Templates := "SrcType := Real" } GE_Contact(in1 := "Conveyor Scale 1 Weight (V)", in2 := 4.0)
      wire#w1
      Contact( "_Retroreflective Sensor 3 package" )
      Coil( "M30.0" )
   END_RUNG
   RUNG wire#powerrail
      Contact( "_FactoryIORunning" )
      Contact( "M30.0" )
   END_RUNG wire#w1
   // the same network as SCL:
   "M30.0" := (("_FactoryIORunning" AND NOT "_Conveyor Scale 1 (+)" AND ("Conveyor Scale 1 Weight (V)" >= 4.0)) OR ("_FactoryIORunning" AND "M30.0")) AND "_Retroreflective Sensor 3 package";
END_REGION

REGION Network 9
   // box M załączenie rolek wraz ze zmianą ich pozycji na 2 sek.
   "IEC_Timer_0_DB".TP(IN := "_FactoryIORunning" AND "M30.0", PT := T#2s);
   "pop_up_box_M" := "IEC_Timer_0_DB".Q;
END_REGION

REGION Network 10
   // załaczenie tasmy przed spadem - warunek
   RUNG wire#powerrail
      Contact( "_FactoryIORunning" )
      wire#w1
      Contact( "M30.0" )
      wire#w2
      Contact( "_Retroreflective Sensor spad" )
      Coil( "M30.2" )
   END_RUNG
   RUNG wire#w1
      Contact( "M30.2" )
   END_RUNG wire#w2
   // the same network as SCL:
   "M30.2" := "_FactoryIORunning" AND ("M30.0" OR "M30.2") AND "_Retroreflective Sensor spad";
END_REGION

REGION Network 11
   RUNG wire#powerrail
      { S7_Templates := "SrcType := Int" } GT_Contact(in1 := "boxes_number_package", in2 := 2)
      Move(in := 2, out1 => "boxes_number_package")
   END_RUNG
   // the same network as SCL:
   IF "boxes_number_package" > 2 THEN "boxes_number_package" := 2; END_IF;
END_REGION

REGION Network 12
   // obliczanie ilosci paczek dla sekcji 1
   #_w1 := "_Retroreflective Sensor spad" AND NOT #mem3;   // rising edge of "_Retroreflective Sensor spad"
   #mem3 := "_Retroreflective Sensor spad";
   "licznik_sekcja_I".CTU(CU := #_w1, R := "_FactoryIOReset", PV := 54);
END_REGION

REGION Network 13
   // przesłanie sygnału o pełnym box'ie
   #_w1 := "_Retroreflective Sensor spad" AND NOT #mem4;   // rising edge of "_Retroreflective Sensor spad"
   #mem4 := "_Retroreflective Sensor spad";
   "IEC_Counter_0_DB".CTU(CU := #_w1,
                          R := ("_Conveyor_sec1_1" AND "Conveyor_sec1_1_Retroreflective Sensor") OR "_FactoryIOReset",
                          PV := "boxes_number_package");
   "box_full" := "IEC_Counter_0_DB".Q;
END_REGION

REGION Network 14
   // zalaczenie tasmy,aby box dojechal po odbior paczki
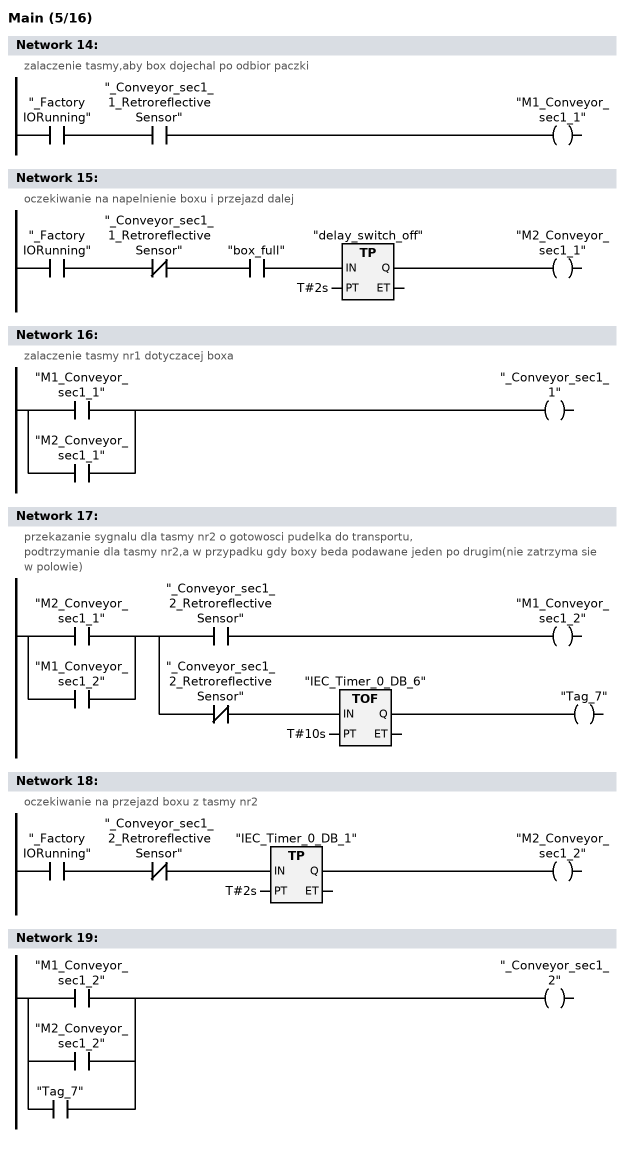
   RUNG wire#powerrail
      Contact( "_FactoryIORunning" )
      Contact( "_Conveyor_sec1_1_Retroreflective Sensor" )
      Coil( "M1_Conveyor_sec1_1" )
   END_RUNG
   // the same network as SCL:
   "M1_Conveyor_sec1_1" := "_FactoryIORunning" AND "_Conveyor_sec1_1_Retroreflective Sensor";
END_REGION

REGION Network 15
   // oczekiwanie na napelnienie boxu i przejazd dalej
   "delay_switch_off".TP(IN := "_FactoryIORunning" AND NOT "_Conveyor_sec1_1_Retroreflective Sensor" AND "box_full",
                         PT := T#2s);
   "M2_Conveyor_sec1_1" := "delay_switch_off".Q;
END_REGION

REGION Network 16
   // zalaczenie tasmy nr1 dotyczacej boxa
   RUNG wire#powerrail
      Contact( "M1_Conveyor_sec1_1" )
      wire#w1
      Coil( "_Conveyor_sec1_1" )
   END_RUNG
   RUNG wire#powerrail
      Contact( "M2_Conveyor_sec1_1" )
   END_RUNG wire#w1
   // the same network as SCL:
   "_Conveyor_sec1_1" := "M1_Conveyor_sec1_1" OR "M2_Conveyor_sec1_1";
END_REGION

REGION Network 17
   // przekazanie sygnalu dla tasmy nr2 o gotowosci pudelka do transportu, 
   // podtrzymanie dla tasmy nr2,a w przypadku gdy boxy beda podawane jeden po drugim(nie zatrzyma sie w polowie)
   #_w1 := "M2_Conveyor_sec1_1" OR "M1_Conveyor_sec1_2";
   "M1_Conveyor_sec1_2" := #_w1 AND "_Conveyor_sec1_2_Retroreflective Sensor";
   "IEC_Timer_0_DB_6".TOF(IN := #_w1 AND NOT "_Conveyor_sec1_2_Retroreflective Sensor", PT := T#10s);
   "Tag_7" := "IEC_Timer_0_DB_6".Q;
END_REGION

REGION Network 18
   // oczekiwanie na przejazd boxu z tasmy nr2
   "IEC_Timer_0_DB_1".TP(IN := "_FactoryIORunning" AND NOT "_Conveyor_sec1_2_Retroreflective Sensor",
                         PT := T#2s);
   "M2_Conveyor_sec1_2" := "IEC_Timer_0_DB_1".Q;
END_REGION

REGION Network 19
   RUNG wire#powerrail
      Contact( "M1_Conveyor_sec1_2" )
      wire#w1
      Coil( "_Conveyor_sec1_2" )
   END_RUNG
   RUNG wire#powerrail
      Contact( "M2_Conveyor_sec1_2" )
   END_RUNG wire#w1
   RUNG wire#powerrail
      Contact( "Tag_7" )
   END_RUNG wire#w1
   // the same network as SCL:
   "_Conveyor_sec1_2" := "M1_Conveyor_sec1_2" OR "M2_Conveyor_sec1_2" OR "Tag_7";
END_REGION

REGION Network 20
   // przekazanie sygnalu dla tasmy nr3 o gotowosci pudelka do transportu
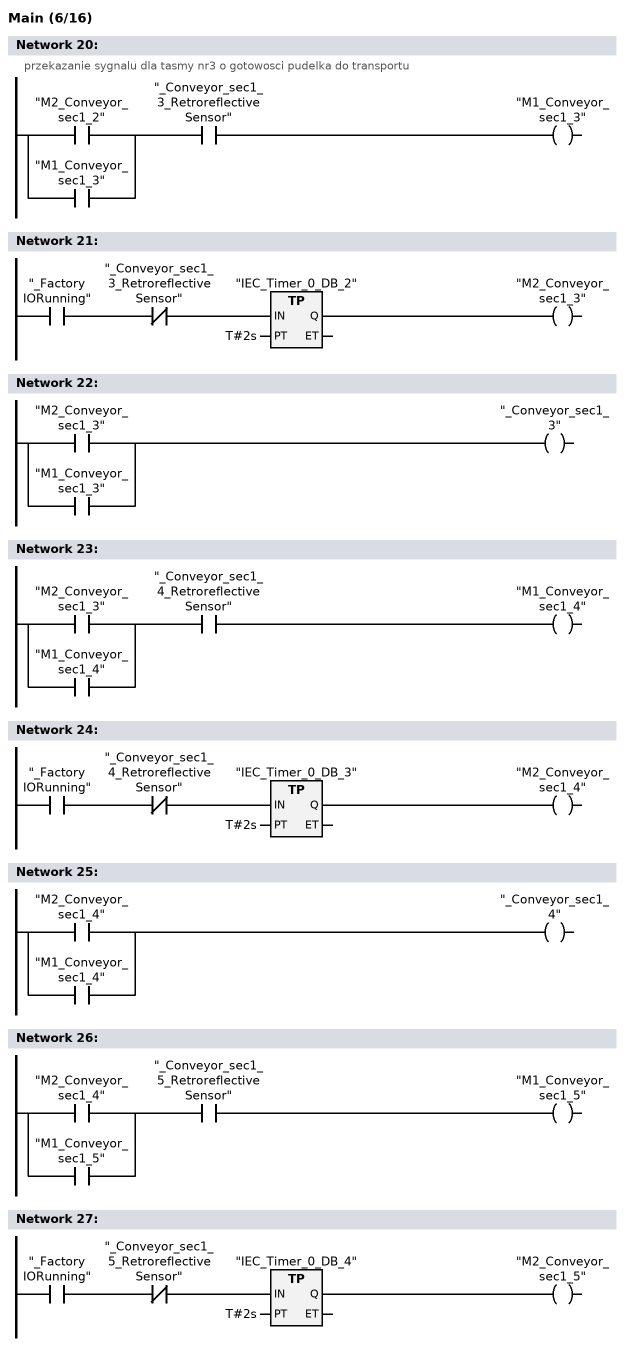
   RUNG wire#powerrail
      Contact( "M2_Conveyor_sec1_2" )
      wire#w1
      Contact( "_Conveyor_sec1_3_Retroreflective Sensor" )
      Coil( "M1_Conveyor_sec1_3" )
   END_RUNG
   RUNG wire#powerrail
      Contact( "M1_Conveyor_sec1_3" )
   END_RUNG wire#w1
   // the same network as SCL:
   "M1_Conveyor_sec1_3" := ("M2_Conveyor_sec1_2" OR "M1_Conveyor_sec1_3") AND "_Conveyor_sec1_3_Retroreflective Sensor";
END_REGION

REGION Network 21
   "IEC_Timer_0_DB_2".TP(IN := "_FactoryIORunning" AND NOT "_Conveyor_sec1_3_Retroreflective Sensor",
                         PT := T#2s);
   "M2_Conveyor_sec1_3" := "IEC_Timer_0_DB_2".Q;
END_REGION

REGION Network 22
   RUNG wire#powerrail
      Contact( "M2_Conveyor_sec1_3" )
      wire#w1
      Coil( "_Conveyor_sec1_3" )
   END_RUNG
   RUNG wire#powerrail
      Contact( "M1_Conveyor_sec1_3" )
   END_RUNG wire#w1
   // the same network as SCL:
   "_Conveyor_sec1_3" := "M2_Conveyor_sec1_3" OR "M1_Conveyor_sec1_3";
END_REGION

REGION Network 23
   RUNG wire#powerrail
      Contact( "M2_Conveyor_sec1_3" )
      wire#w1
      Contact( "_Conveyor_sec1_4_Retroreflective Sensor" )
      Coil( "M1_Conveyor_sec1_4" )
   END_RUNG
   RUNG wire#powerrail
      Contact( "M1_Conveyor_sec1_4" )
   END_RUNG wire#w1
   // the same network as SCL:
   "M1_Conveyor_sec1_4" := ("M2_Conveyor_sec1_3" OR "M1_Conveyor_sec1_4") AND "_Conveyor_sec1_4_Retroreflective Sensor";
END_REGION

REGION Network 24
   "IEC_Timer_0_DB_3".TP(IN := "_FactoryIORunning" AND NOT "_Conveyor_sec1_4_Retroreflective Sensor",
                         PT := T#2s);
   "M2_Conveyor_sec1_4" := "IEC_Timer_0_DB_3".Q;
END_REGION

REGION Network 25
   RUNG wire#powerrail
      Contact( "M2_Conveyor_sec1_4" )
      wire#w1
      Coil( "_Conveyor_sec1_4" )
   END_RUNG
   RUNG wire#powerrail
      Contact( "M1_Conveyor_sec1_4" )
   END_RUNG wire#w1
   // the same network as SCL:
   "_Conveyor_sec1_4" := "M2_Conveyor_sec1_4" OR "M1_Conveyor_sec1_4";
END_REGION

REGION Network 26
   RUNG wire#powerrail
      Contact( "M2_Conveyor_sec1_4" )
      wire#w1
      Contact( "_Conveyor_sec1_5_Retroreflective Sensor" )
      Coil( "M1_Conveyor_sec1_5" )
   END_RUNG
   RUNG wire#powerrail
      Contact( "M1_Conveyor_sec1_5" )
   END_RUNG wire#w1
   // the same network as SCL:
   "M1_Conveyor_sec1_5" := ("M2_Conveyor_sec1_4" OR "M1_Conveyor_sec1_5") AND "_Conveyor_sec1_5_Retroreflective Sensor";
END_REGION

REGION Network 27
   "IEC_Timer_0_DB_4".TP(IN := "_FactoryIORunning" AND NOT "_Conveyor_sec1_5_Retroreflective Sensor",
                         PT := T#2s);
   "M2_Conveyor_sec1_5" := "IEC_Timer_0_DB_4".Q;
END_REGION

REGION Network 28
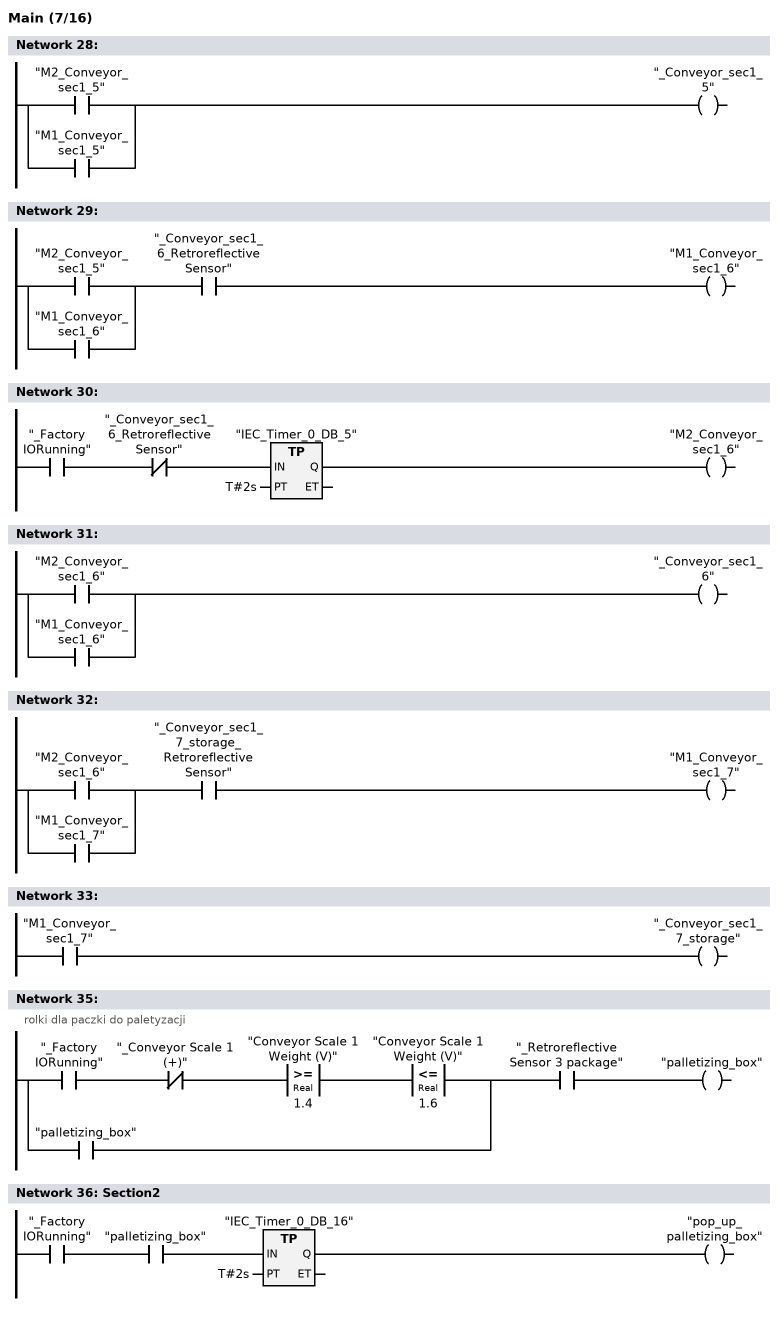
   RUNG wire#powerrail
      Contact( "M2_Conveyor_sec1_5" )
      wire#w1
      Coil( "_Conveyor_sec1_5" )
   END_RUNG
   RUNG wire#powerrail
      Contact( "M1_Conveyor_sec1_5" )
   END_RUNG wire#w1
   // the same network as SCL:
   "_Conveyor_sec1_5" := "M2_Conveyor_sec1_5" OR "M1_Conveyor_sec1_5";
END_REGION

REGION Network 29
   RUNG wire#powerrail
      Contact( "M2_Conveyor_sec1_5" )
      wire#w1
      Contact( "_Conveyor_sec1_6_Retroreflective Sensor" )
      Coil( "M1_Conveyor_sec1_6" )
   END_RUNG
   RUNG wire#powerrail
      Contact( "M1_Conveyor_sec1_6" )
   END_RUNG wire#w1
   // the same network as SCL:
   "M1_Conveyor_sec1_6" := ("M2_Conveyor_sec1_5" OR "M1_Conveyor_sec1_6") AND "_Conveyor_sec1_6_Retroreflective Sensor";
END_REGION

REGION Network 30
   "IEC_Timer_0_DB_5".TP(IN := "_FactoryIORunning" AND NOT "_Conveyor_sec1_6_Retroreflective Sensor",
                         PT := T#2s);
   "M2_Conveyor_sec1_6" := "IEC_Timer_0_DB_5".Q;
END_REGION

REGION Network 31
   RUNG wire#powerrail
      Contact( "M2_Conveyor_sec1_6" )
      wire#w1
      Coil( "_Conveyor_sec1_6" )
   END_RUNG
   RUNG wire#powerrail
      Contact( "M1_Conveyor_sec1_6" )
   END_RUNG wire#w1
   // the same network as SCL:
   "_Conveyor_sec1_6" := "M2_Conveyor_sec1_6" OR "M1_Conveyor_sec1_6";
END_REGION

REGION Network 32
   RUNG wire#powerrail
      Contact( "M2_Conveyor_sec1_6" )
      wire#w1
      Contact( "_Conveyor_sec1_7_storage_Retroreflective Sensor" )
      Coil( "M1_Conveyor_sec1_7" )
   END_RUNG
   RUNG wire#powerrail
      Contact( "M1_Conveyor_sec1_7" )
   END_RUNG wire#w1
   // the same network as SCL:
   "M1_Conveyor_sec1_7" := ("M2_Conveyor_sec1_6" OR "M1_Conveyor_sec1_7") AND "_Conveyor_sec1_7_storage_Retroreflective Sensor";
END_REGION

REGION Network 33
   RUNG wire#powerrail
      Contact( "M1_Conveyor_sec1_7" )
      Coil( "_Conveyor_sec1_7_storage" )
   END_RUNG
   // the same network as SCL:
   "_Conveyor_sec1_7_storage" := "M1_Conveyor_sec1_7";
END_REGION

REGION Network 35
   // rolki dla paczki do paletyzacji
   RUNG wire#powerrail
      Contact( "_FactoryIORunning" )
      I_Contact( "_Conveyor Scale 1 (+)" )
      { S7_Templates := "SrcType := Real" } GE_Contact(in1 := "Conveyor Scale 1 Weight (V)", in2 := 1.4)
      { S7_Templates := "SrcType := Real" } LE_Contact(in1 := "Conveyor Scale 1 Weight (V)", in2 := 1.6)
      wire#w1
      Contact( "_Retroreflective Sensor 3 package" )
      Coil( "palletizing_box" )
   END_RUNG
   RUNG wire#powerrail
      Contact( "palletizing_box" )
   END_RUNG wire#w1
   // the same network as SCL:
   "palletizing_box" := (("_FactoryIORunning" AND NOT "_Conveyor Scale 1 (+)" AND ("Conveyor Scale 1 Weight (V)" >= 1.4) AND ("Conveyor Scale 1 Weight (V)" <= 1.6)) OR "palletizing_box") AND "_Retroreflective Sensor 3 package";
END_REGION

REGION Network 36: Section2
   "IEC_Timer_0_DB_16".TP(IN := "_FactoryIORunning" AND "palletizing_box", PT := T#2s);
   "pop_up_palletizing_box" := "IEC_Timer_0_DB_16".Q;
END_REGION

REGION Network 37
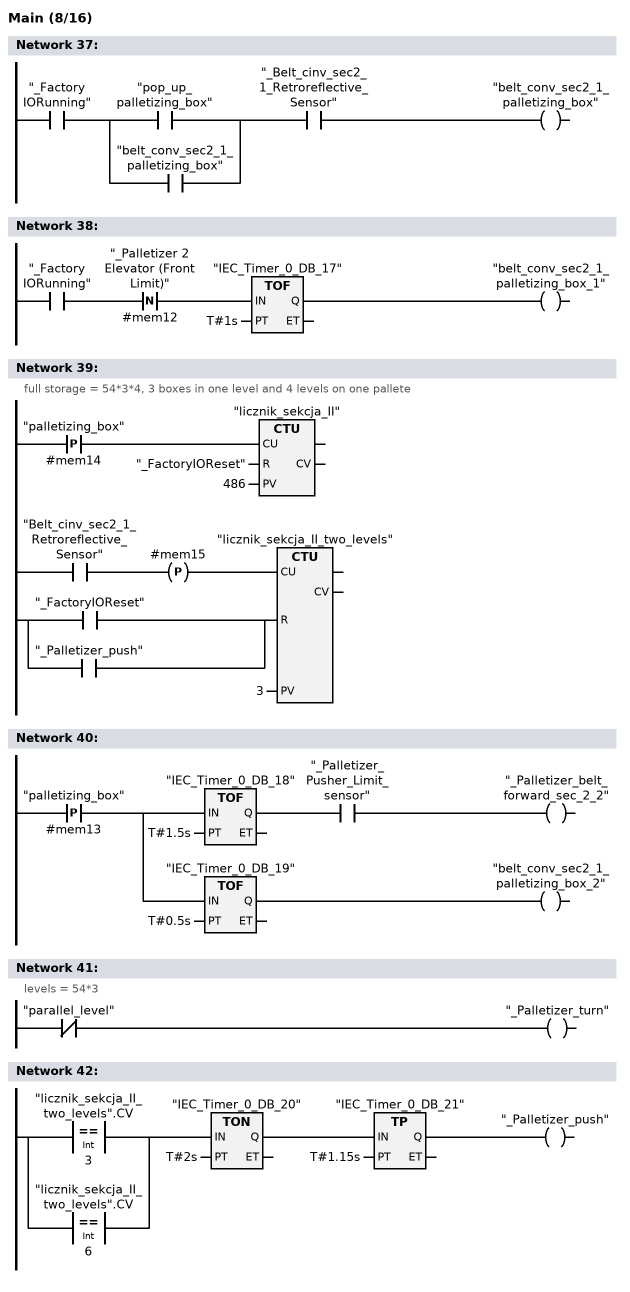
   RUNG wire#powerrail
      Contact( "_FactoryIORunning" )
      wire#w1
      Contact( "pop_up_palletizing_box" )
      wire#w2
      Contact( "_Belt_cinv_sec2_1_Retroreflective_Sensor" )
      Coil( "belt_conv_sec2_1_palletizing_box" )
   END_RUNG
   RUNG wire#w1
      Contact( "belt_conv_sec2_1_palletizing_box" )
   END_RUNG wire#w2
   // the same network as SCL:
   "belt_conv_sec2_1_palletizing_box" := "_FactoryIORunning" AND ("pop_up_palletizing_box" OR "belt_conv_sec2_1_palletizing_box") AND "_Belt_cinv_sec2_1_Retroreflective_Sensor";
END_REGION

REGION Network 38
   #_w1 := "_FactoryIORunning" AND NOT "_Palletizer 2 Elevator (Front Limit)" AND #mem12;   // falling edge of "_Palletizer 2 Elevator (Front Limit)"
   #mem12 := "_Palletizer 2 Elevator (Front Limit)";
   "IEC_Timer_0_DB_17".TOF(IN := #_w1, PT := T#1s);
   "belt_conv_sec2_1_palletizing_box_1" := "IEC_Timer_0_DB_17".Q;
END_REGION

REGION Network 39
   // full storage = 54*3*4, 3 boxes in one level and 4 levels on one pallete
   #_w1 := "palletizing_box" AND NOT #mem14;   // rising edge of "palletizing_box"
   #mem14 := "palletizing_box";
   "licznik_sekcja_II".CTU(CU := #_w1, R := "_FactoryIOReset", PV := 486);
   #_w2 := "Belt_cinv_sec2_1_Retroreflective_Sensor" AND NOT #mem15;   // rising edge
   #mem15 := "Belt_cinv_sec2_1_Retroreflective_Sensor";
   "licznik_sekcja_II_two_levels".CTU(CU := #_w2, R := "_FactoryIOReset" OR "_Palletizer_push", PV := 3);
END_REGION

REGION Network 40
   #_w1 := "palletizing_box" AND NOT #mem13;   // rising edge of "palletizing_box"
   #mem13 := "palletizing_box";
   "IEC_Timer_0_DB_18".TOF(IN := #_w1, PT := T#1.5s);
   "_Palletizer_belt_forward_sec_2_2" := "IEC_Timer_0_DB_18".Q AND "_Palletizer_Pusher_Limit_sensor";
   "IEC_Timer_0_DB_19".TOF(IN := #_w1, PT := T#0.5s);
   "belt_conv_sec2_1_palletizing_box_2" := "IEC_Timer_0_DB_19".Q;
END_REGION

REGION Network 41
   // levels = 54*3
   RUNG wire#powerrail
      I_Contact( "parallel_level" )
      Coil( "_Palletizer_turn" )
   END_RUNG
   // the same network as SCL:
   "_Palletizer_turn" := NOT "parallel_level";
END_REGION

REGION Network 42
   "IEC_Timer_0_DB_20".TON(IN := ("licznik_sekcja_II_two_levels".CV = 3) OR ("licznik_sekcja_II_two_levels".CV = 6),
                           PT := T#2s);
   "IEC_Timer_0_DB_21".TP(IN := "IEC_Timer_0_DB_20".Q, PT := T#1.15s);
   "_Palletizer_push" := "IEC_Timer_0_DB_21".Q;
END_REGION

REGION Network 43
   // turn boxes
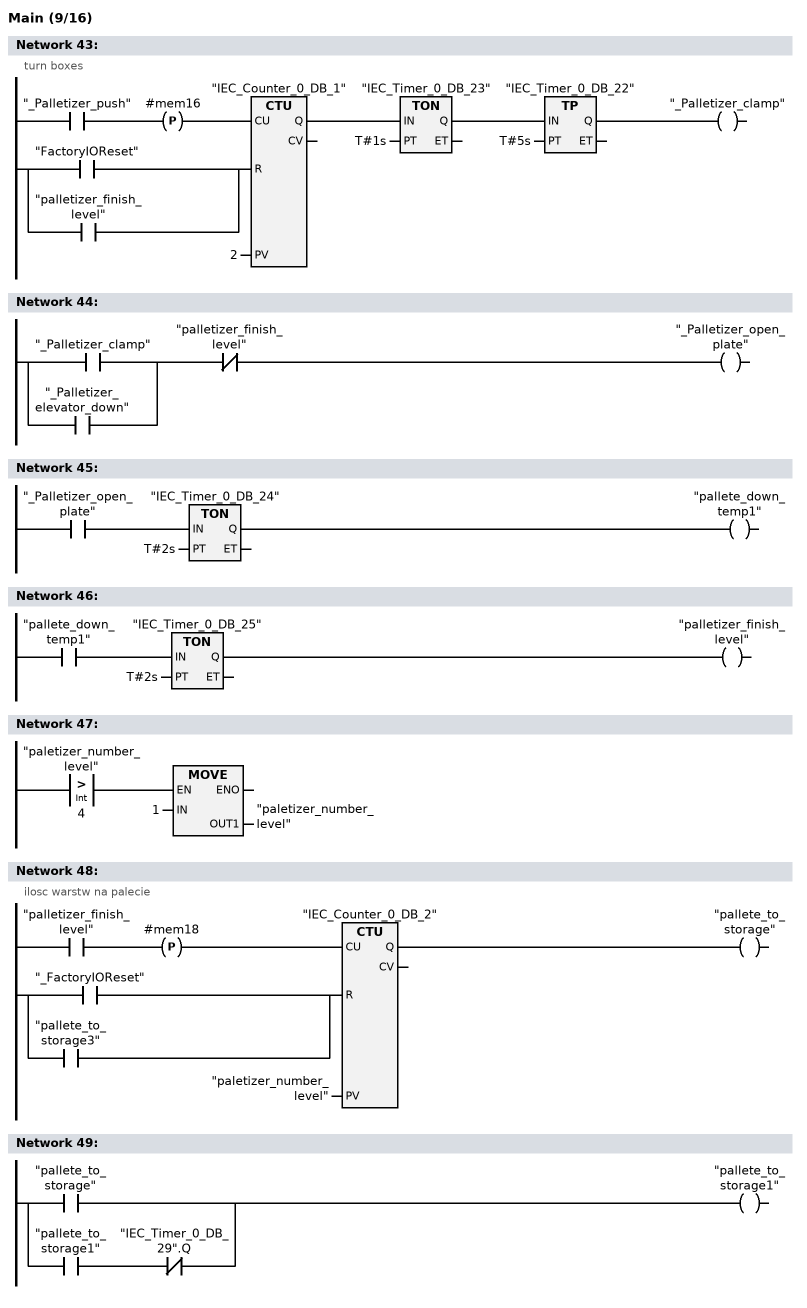
   #_w1 := "_Palletizer_push" AND NOT #mem16;   // rising edge
   #mem16 := "_Palletizer_push";
   "IEC_Counter_0_DB_1".CTU(CU := #_w1, R := "FactoryIOReset" OR "palletizer_finish_level", PV := 2);
   "IEC_Timer_0_DB_23".TON(IN := "IEC_Counter_0_DB_1".Q, PT := T#1s);
   "IEC_Timer_0_DB_22".TP(IN := "IEC_Timer_0_DB_23".Q, PT := T#5s);
   "_Palletizer_clamp" := "IEC_Timer_0_DB_22".Q;
END_REGION

REGION Network 44
   RUNG wire#powerrail
      Contact( "_Palletizer_clamp" )
      wire#w1
      I_Contact( "palletizer_finish_level" )
      Coil( "_Palletizer_open_plate" )
   END_RUNG
   RUNG wire#powerrail
      Contact( "_Palletizer_elevator_down" )
   END_RUNG wire#w1
   // the same network as SCL:
   "_Palletizer_open_plate" := ("_Palletizer_clamp" OR "_Palletizer_elevator_down") AND NOT "palletizer_finish_level";
END_REGION

REGION Network 45
   "IEC_Timer_0_DB_24".TON(IN := "_Palletizer_open_plate", PT := T#2s);
   "pallete_down_temp1" := "IEC_Timer_0_DB_24".Q;
END_REGION

REGION Network 46
   "IEC_Timer_0_DB_25".TON(IN := "pallete_down_temp1", PT := T#2s);
   "palletizer_finish_level" := "IEC_Timer_0_DB_25".Q;
END_REGION

REGION Network 47
   RUNG wire#powerrail
      { S7_Templates := "SrcType := Int" } GT_Contact(in1 := "paletizer_number_level", in2 := 4)
      Move(in := 1, out1 => "paletizer_number_level")
   END_RUNG
   // the same network as SCL:
   IF "paletizer_number_level" > 4 THEN "paletizer_number_level" := 1; END_IF;
END_REGION

REGION Network 48
   // ilosc warstw na palecie
   #_w1 := "palletizer_finish_level" AND NOT #mem18;   // rising edge
   #mem18 := "palletizer_finish_level";
   "IEC_Counter_0_DB_2".CTU(CU := #_w1,
                           R := "_FactoryIOReset" OR "pallete_to_storage3",
                           PV := "paletizer_number_level");
   "pallete_to_storage" := "IEC_Counter_0_DB_2".Q;
END_REGION

REGION Network 49
   RUNG wire#powerrail
      Contact( "pallete_to_storage" )
      wire#w1
      Coil( "pallete_to_storage1" )
   END_RUNG
   RUNG wire#powerrail
      Contact( "pallete_to_storage1" )
      I_Contact( "IEC_Timer_0_DB_29".Q )
   END_RUNG wire#w1
   // the same network as SCL:
   "pallete_to_storage1" := "pallete_to_storage" OR ("pallete_to_storage1" AND NOT "IEC_Timer_0_DB_29".Q);
END_REGION

REGION Network 50
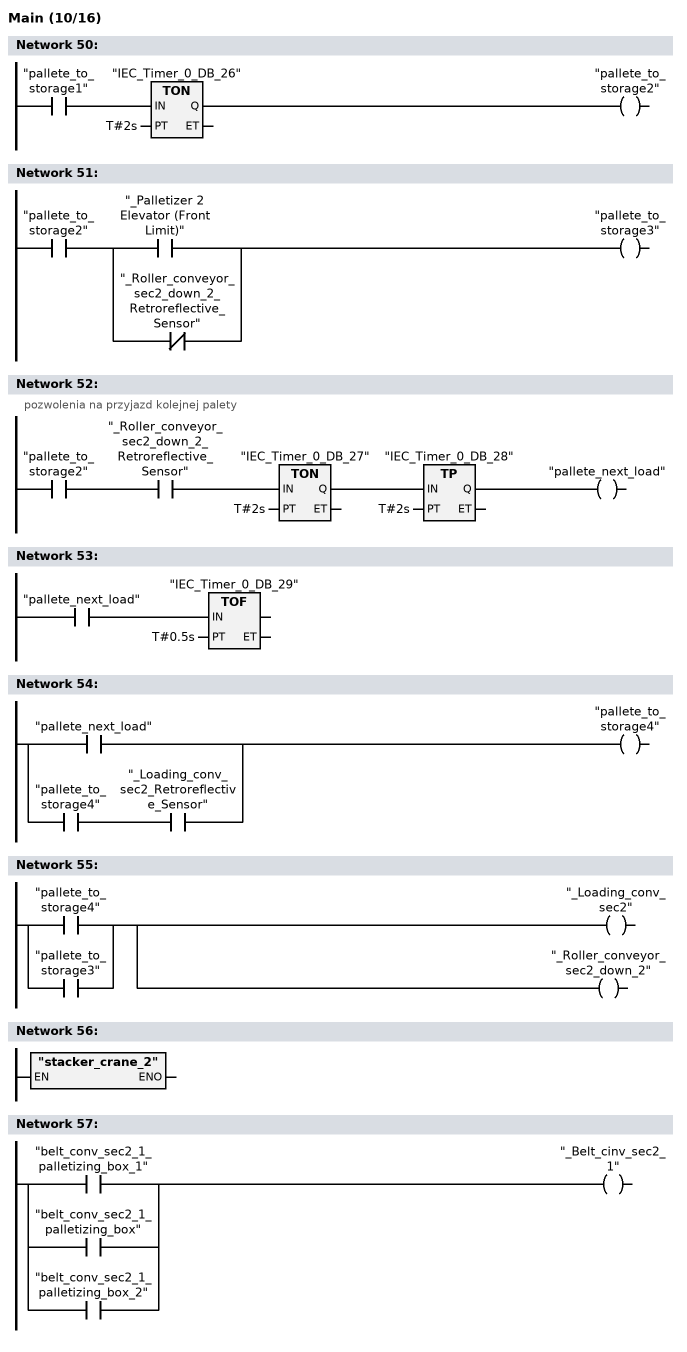
   "IEC_Timer_0_DB_26".TON(IN := "pallete_to_storage1", PT := T#2s);
   "pallete_to_storage2" := "IEC_Timer_0_DB_26".Q;
END_REGION

REGION Network 51
   RUNG wire#powerrail
      Contact( "pallete_to_storage2" )
      wire#w1
      Contact( "_Palletizer 2 Elevator (Front Limit)" )
      wire#w2
      Coil( "pallete_to_storage3" )
   END_RUNG
   RUNG wire#w1
      I_Contact( "_Roller_conveyor_sec2_down_2_Retroreflective_Sensor" )
   END_RUNG wire#w2
   // the same network as SCL:
   "pallete_to_storage3" := "pallete_to_storage2" AND ("_Palletizer 2 Elevator (Front Limit)" OR NOT "_Roller_conveyor_sec2_down_2_Retroreflective_Sensor");
END_REGION

REGION Network 52
   // pozwolenia na przyjazd kolejnej palety
   "IEC_Timer_0_DB_27".TON(IN := "pallete_to_storage2" AND "_Roller_conveyor_sec2_down_2_Retroreflective_Sensor",
                           PT := T#2s);
   "IEC_Timer_0_DB_28".TP(IN := "IEC_Timer_0_DB_27".Q, PT := T#2s);
   "pallete_next_load" := "IEC_Timer_0_DB_28".Q;
END_REGION

REGION Network 53
   "IEC_Timer_0_DB_29".TOF(IN := "pallete_next_load", PT := T#0.5s);
END_REGION

REGION Network 54
   RUNG wire#powerrail
      Contact( "pallete_next_load" )
      wire#w1
      Coil( "pallete_to_storage4" )
   END_RUNG
   RUNG wire#powerrail
      Contact( "pallete_to_storage4" )
      Contact( "_Loading_conv_sec2_Retroreflective_Sensor" )
   END_RUNG wire#w1
   // the same network as SCL:
   "pallete_to_storage4" := "pallete_next_load" OR ("pallete_to_storage4" AND "_Loading_conv_sec2_Retroreflective_Sensor");
END_REGION

REGION Network 55
   RUNG wire#powerrail
      Contact( "pallete_to_storage4" )
      wire#w1
      Coil( "_Loading_conv_sec2" )
   END_RUNG
   RUNG wire#powerrail
      Contact( "pallete_to_storage3" )
   END_RUNG wire#w1
   RUNG wire#w1
      Coil( "_Roller_conveyor_sec2_down_2" )
   END_RUNG
   // the same network as SCL:
   "_Loading_conv_sec2" := "pallete_to_storage4" OR "pallete_to_storage3";
   "_Roller_conveyor_sec2_down_2" := "_Loading_conv_sec2";
END_REGION

REGION Network 56
   RUNG wire#powerrail
      "stacker_crane_2"()
   END_RUNG
   // the same network as SCL:
   "stacker_crane_2"();
END_REGION

REGION Network 57
   RUNG wire#powerrail
      Contact( "belt_conv_sec2_1_palletizing_box_1" )
      wire#w1
      Coil( "_Belt_cinv_sec2_1" )
   END_RUNG
   RUNG wire#powerrail
      Contact( "belt_conv_sec2_1_palletizing_box" )
   END_RUNG wire#w1
   RUNG wire#powerrail
      Contact( "belt_conv_sec2_1_palletizing_box_2" )
   END_RUNG wire#w1
   // the same network as SCL:
   "_Belt_cinv_sec2_1" := "belt_conv_sec2_1_palletizing_box_1" OR "belt_conv_sec2_1_palletizing_box" OR "belt_conv_sec2_1_palletizing_box_2";
END_REGION

REGION Network 60
   // obsluga rozmiaru paczek
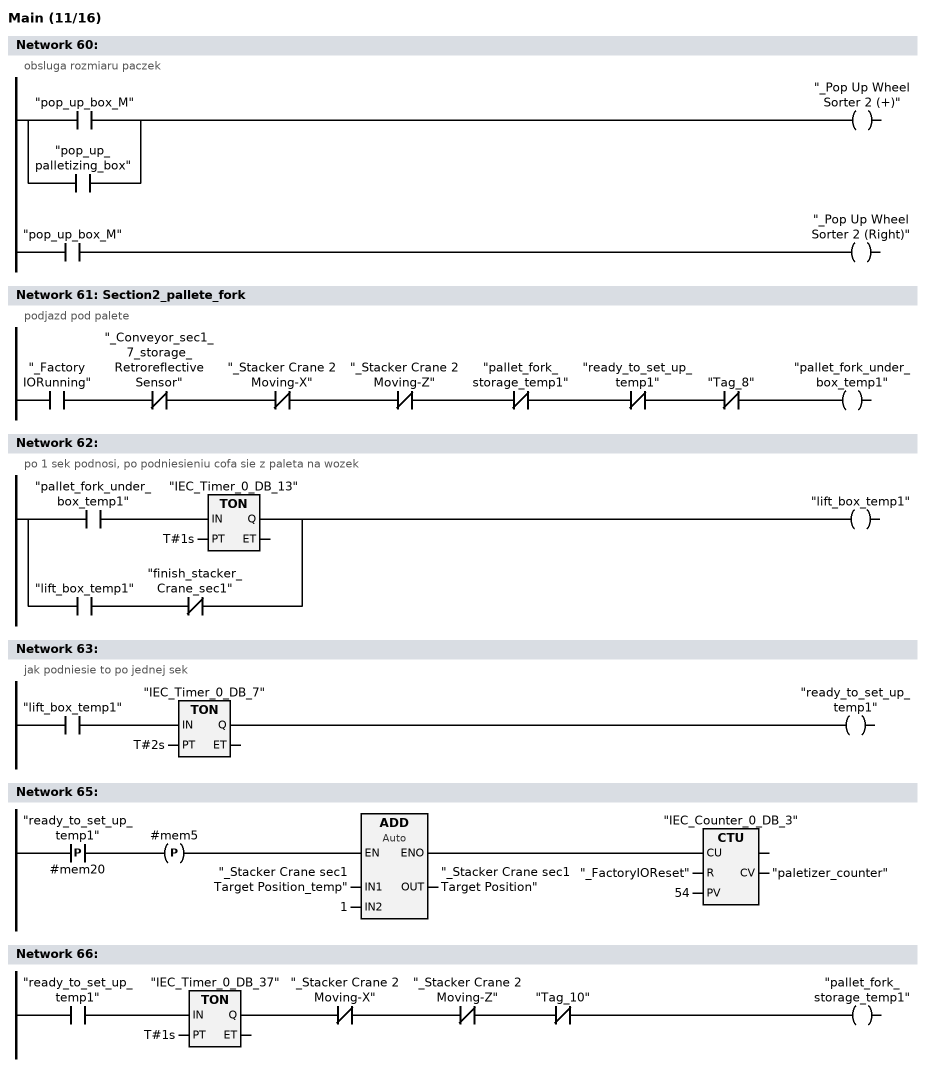
   RUNG wire#powerrail
      Contact( "pop_up_box_M" )
      wire#w1
      Coil( "_Pop Up Wheel Sorter 2 (+)" )
   END_RUNG
   RUNG wire#powerrail
      Contact( "pop_up_palletizing_box" )
   END_RUNG wire#w1
   RUNG wire#powerrail
      Contact( "pop_up_box_M" )
      Coil( "_Pop Up Wheel Sorter 2 (Right)" )
   END_RUNG
   // the same network as SCL:
   "_Pop Up Wheel Sorter 2 (+)" := "pop_up_box_M" OR "pop_up_palletizing_box";
   "_Pop Up Wheel Sorter 2 (Right)" := "pop_up_box_M";
END_REGION

REGION Network 61: Section2_pallete_fork
   // podjazd pod palete
   RUNG wire#powerrail
      Contact( "_FactoryIORunning" )
      I_Contact( "_Conveyor_sec1_7_storage_Retroreflective Sensor" )
      I_Contact( "_Stacker Crane 2 Moving-X" )
      I_Contact( "_Stacker Crane 2 Moving-Z" )
      I_Contact( "pallet_fork_storage_temp1" )
      I_Contact( "ready_to_set_up_temp1" )
      I_Contact( "Tag_8" )
      Coil( "pallet_fork_under_box_temp1" )
   END_RUNG
   // the same network as SCL:
   "pallet_fork_under_box_temp1" := "_FactoryIORunning" AND NOT "_Conveyor_sec1_7_storage_Retroreflective Sensor" AND NOT "_Stacker Crane 2 Moving-X" AND NOT "_Stacker Crane 2 Moving-Z" AND NOT "pallet_fork_storage_temp1" AND NOT "ready_to_set_up_temp1" AND NOT "Tag_8";
END_REGION

REGION Network 62
   // po 1 sek podnosi, po podniesieniu cofa sie z paleta na wozek
   "IEC_Timer_0_DB_13".TON(IN := "pallet_fork_under_box_temp1", PT := T#1s);
   "lift_box_temp1" := "IEC_Timer_0_DB_13".Q OR ("lift_box_temp1" AND NOT "finish_stacker_Crane_sec1");
END_REGION

REGION Network 63
   // jak podniesie to po jednej sek
   "IEC_Timer_0_DB_7".TON(IN := "lift_box_temp1", PT := T#2s);
   "ready_to_set_up_temp1" := "IEC_Timer_0_DB_7".Q;
END_REGION

REGION Network 65
   #_w1 := "ready_to_set_up_temp1" AND NOT #mem20;   // rising edge of "ready_to_set_up_temp1"
   #mem20 := "ready_to_set_up_temp1";
   #_w2 := #_w1 AND NOT #mem5;   // rising edge
   #mem5 := #_w1;
   IF #_w2 THEN
       "_Stacker Crane sec1 Target Position" := "_Stacker Crane sec1 Target Position_temp" + 1;
   END_IF;
   "IEC_Counter_0_DB_3".CTU(CU := #_w2, R := "_FactoryIOReset", PV := 54, CV => "paletizer_counter");
END_REGION

REGION Network 66
   "IEC_Timer_0_DB_37".TON(IN := "ready_to_set_up_temp1", PT := T#1s);
   "pallet_fork_storage_temp1" := "IEC_Timer_0_DB_37".Q AND NOT "_Stacker Crane 2 Moving-X" AND NOT "_Stacker Crane 2 Moving-Z" AND NOT "Tag_10";
END_REGION

REGION Network 67
   // opuszczanie po 1sek
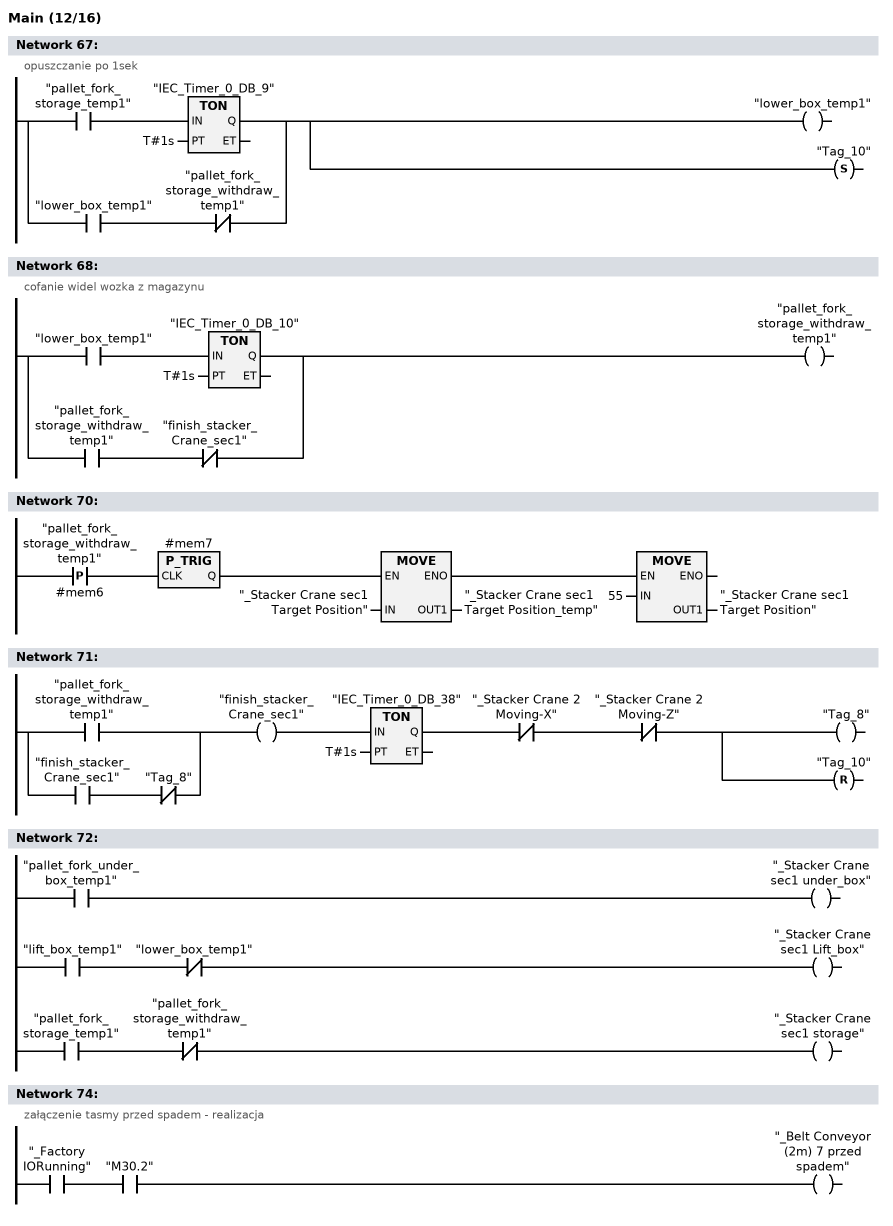
   "IEC_Timer_0_DB_9".TON(IN := "pallet_fork_storage_temp1", PT := T#1s);
   "lower_box_temp1" := "IEC_Timer_0_DB_9".Q OR ("lower_box_temp1" AND NOT "pallet_fork_storage_withdraw_temp1");
   IF "lower_box_temp1" THEN "Tag_10" := TRUE; END_IF;
END_REGION

REGION Network 68
   // cofanie widel wozka z magazynu
   "IEC_Timer_0_DB_10".TON(IN := "lower_box_temp1", PT := T#1s);
   "pallet_fork_storage_withdraw_temp1" := "IEC_Timer_0_DB_10".Q OR ("pallet_fork_storage_withdraw_temp1" AND NOT "finish_stacker_Crane_sec1");
END_REGION

REGION Network 69
   // powrot na pozycje startowa widlaka
END_REGION

REGION Network 70
   RUNG wire#powerrail
      P_Contact(operand := "pallet_fork_storage_withdraw_temp1", bit := #mem6)
      P_Trig( #mem7 )
      Move(in := "_Stacker Crane sec1 Target Position", out1 => "_Stacker Crane sec1 Target Position_temp")
      Move(in := 55, out1 => "_Stacker Crane sec1 Target Position")
   END_RUNG
   // the same network as SCL:
   #_w1 := "pallet_fork_storage_withdraw_temp1" AND NOT #mem6;   // rising edge of "pallet_fork_storage_withdraw_temp1"
   #mem6 := "pallet_fork_storage_withdraw_temp1";
   #_w2 := #_w1 AND NOT #mem7;   // rising edge
   #mem7 := #_w1;
   IF #_w2 THEN
       "_Stacker Crane sec1 Target Position_temp" := "_Stacker Crane sec1 Target Position";
       "_Stacker Crane sec1 Target Position" := 55;
   END_IF;
END_REGION

REGION Network 71
   "finish_stacker_Crane_sec1" := "pallet_fork_storage_withdraw_temp1" OR ("finish_stacker_Crane_sec1" AND NOT "Tag_8");
   "IEC_Timer_0_DB_38".TON(IN := "finish_stacker_Crane_sec1", PT := T#1s);
   "Tag_8" := "IEC_Timer_0_DB_38".Q AND NOT "_Stacker Crane 2 Moving-X" AND NOT "_Stacker Crane 2 Moving-Z";
   IF "Tag_8" THEN "Tag_10" := FALSE; END_IF;
END_REGION

REGION Network 72
   RUNG wire#powerrail
      Contact( "pallet_fork_under_box_temp1" )
      Coil( "_Stacker Crane sec1 under_box" )
   END_RUNG
   RUNG wire#powerrail
      Contact( "lift_box_temp1" )
      I_Contact( "lower_box_temp1" )
      Coil( "_Stacker Crane sec1 Lift_box" )
   END_RUNG
   RUNG wire#powerrail
      Contact( "pallet_fork_storage_temp1" )
      I_Contact( "pallet_fork_storage_withdraw_temp1" )
      Coil( "_Stacker Crane sec1 storage" )
   END_RUNG
   // the same network as SCL:
   "_Stacker Crane sec1 under_box" := "pallet_fork_under_box_temp1";
   "_Stacker Crane sec1 Lift_box" := "lift_box_temp1" AND NOT "lower_box_temp1";
   "_Stacker Crane sec1 storage" := "pallet_fork_storage_temp1" AND NOT "pallet_fork_storage_withdraw_temp1";
END_REGION

REGION Network 74
   // załączenie tasmy przed spadem - realizacja
   RUNG wire#powerrail
      Contact( "_FactoryIORunning" )
      Contact( "M30.2" )
      Coil( "_Belt Conveyor (2m) 7 przed spadem" )
   END_RUNG
   // the same network as SCL:
   "_Belt Conveyor (2m) 7 przed spadem" := "_FactoryIORunning" AND "M30.2";
END_REGION

REGION Network 75
   // ruch wagi
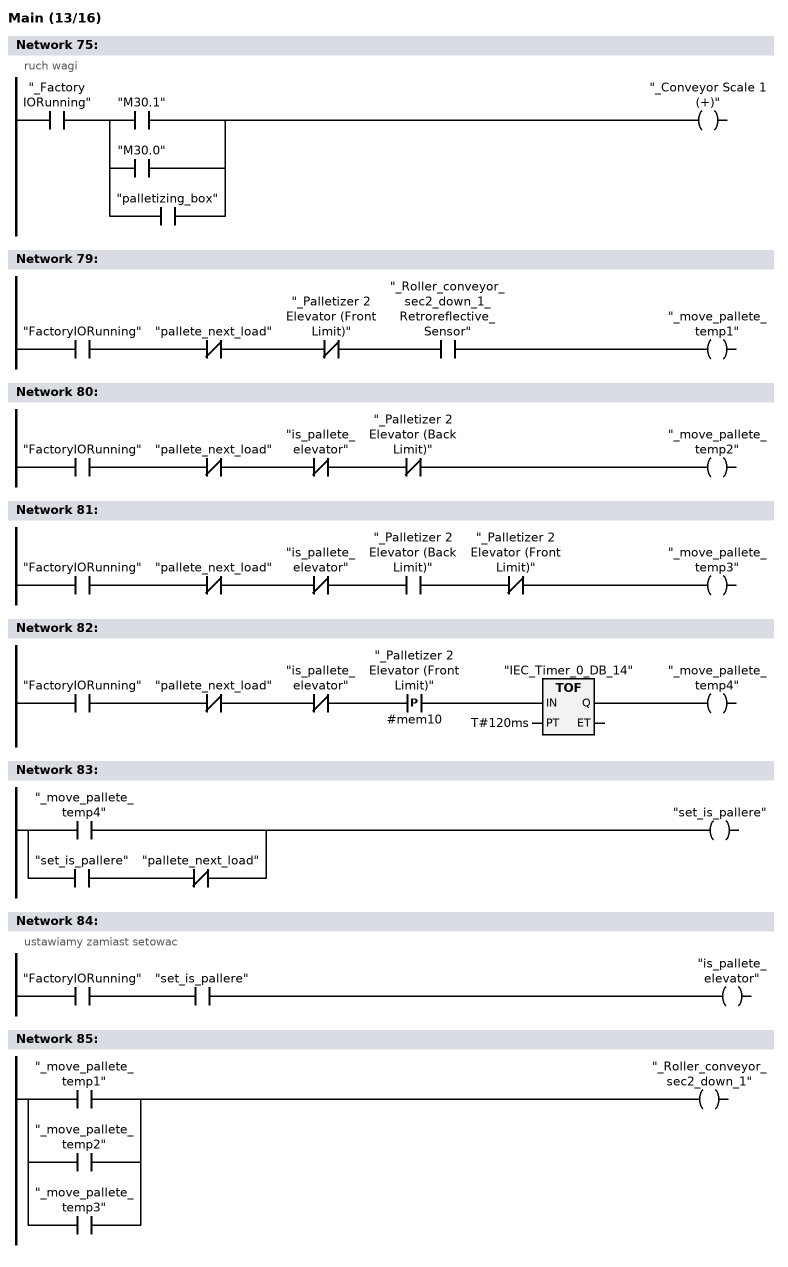
   RUNG wire#powerrail
      Contact( "_FactoryIORunning" )
      wire#w1
      Contact( "M30.1" )
      wire#w2
      Coil( "_Conveyor Scale 1 (+)" )
   END_RUNG
   RUNG wire#w1
      Contact( "M30.0" )
   END_RUNG wire#w2
   RUNG wire#w1
      Contact( "palletizing_box" )
   END_RUNG wire#w2
   // the same network as SCL:
   "_Conveyor Scale 1 (+)" := "_FactoryIORunning" AND ("M30.1" OR "M30.0" OR "palletizing_box");
END_REGION

REGION Network 77: Section 2 - transport wooden pallets
END_REGION

REGION Network 79
   RUNG wire#powerrail
      Contact( "FactoryIORunning" )
      I_Contact( "pallete_next_load" )
      I_Contact( "_Palletizer 2 Elevator (Front Limit)" )
      Contact( "_Roller_conveyor_sec2_down_1_Retroreflective_Sensor" )
      Coil( "_move_pallete_temp1" )
   END_RUNG
   // the same network as SCL:
   "_move_pallete_temp1" := "FactoryIORunning" AND NOT "pallete_next_load" AND NOT "_Palletizer 2 Elevator (Front Limit)" AND "_Roller_conveyor_sec2_down_1_Retroreflective_Sensor";
END_REGION

REGION Network 80
   RUNG wire#powerrail
      Contact( "FactoryIORunning" )
      I_Contact( "pallete_next_load" )
      I_Contact( "is_pallete_elevator" )
      I_Contact( "_Palletizer 2 Elevator (Back Limit)" )
      Coil( "_move_pallete_temp2" )
   END_RUNG
   // the same network as SCL:
   "_move_pallete_temp2" := "FactoryIORunning" AND NOT "pallete_next_load" AND NOT "is_pallete_elevator" AND NOT "_Palletizer 2 Elevator (Back Limit)";
END_REGION

REGION Network 81
   RUNG wire#powerrail
      Contact( "FactoryIORunning" )
      I_Contact( "pallete_next_load" )
      I_Contact( "is_pallete_elevator" )
      Contact( "_Palletizer 2 Elevator (Back Limit)" )
      I_Contact( "_Palletizer 2 Elevator (Front Limit)" )
      Coil( "_move_pallete_temp3" )
   END_RUNG
   // the same network as SCL:
   "_move_pallete_temp3" := "FactoryIORunning" AND NOT "pallete_next_load" AND NOT "is_pallete_elevator" AND "_Palletizer 2 Elevator (Back Limit)" AND NOT "_Palletizer 2 Elevator (Front Limit)";
END_REGION

REGION Network 82
   #_w1 := "FactoryIORunning" AND NOT "pallete_next_load" AND NOT "is_pallete_elevator" AND "_Palletizer 2 Elevator (Front Limit)" AND NOT #mem10;   // rising edge of "_Palletizer 2 Elevator (Front Limit)"
   #mem10 := "_Palletizer 2 Elevator (Front Limit)";
   "IEC_Timer_0_DB_14".TOF(IN := #_w1, PT := T#120ms);
   "_move_pallete_temp4" := "IEC_Timer_0_DB_14".Q;
END_REGION

REGION Network 83
   RUNG wire#powerrail
      Contact( "_move_pallete_temp4" )
      wire#w1
      Coil( "set_is_pallere" )
   END_RUNG
   RUNG wire#powerrail
      Contact( "set_is_pallere" )
      I_Contact( "pallete_next_load" )
   END_RUNG wire#w1
   // the same network as SCL:
   "set_is_pallere" := "_move_pallete_temp4" OR ("set_is_pallere" AND NOT "pallete_next_load");
END_REGION

REGION Network 84
   // ustawiamy zamiast setowac
   RUNG wire#powerrail
      Contact( "FactoryIORunning" )
      Contact( "set_is_pallere" )
      Coil( "is_pallete_elevator" )
   END_RUNG
   // the same network as SCL:
   "is_pallete_elevator" := "FactoryIORunning" AND "set_is_pallere";
END_REGION

REGION Network 85
   RUNG wire#powerrail
      Contact( "_move_pallete_temp1" )
      wire#w1
      Coil( "_Roller_conveyor_sec2_down_1" )
   END_RUNG
   RUNG wire#powerrail
      Contact( "_move_pallete_temp2" )
   END_RUNG wire#w1
   RUNG wire#powerrail
      Contact( "_move_pallete_temp3" )
   END_RUNG wire#w1
   // the same network as SCL:
   "_Roller_conveyor_sec2_down_1" := "_move_pallete_temp1" OR "_move_pallete_temp2" OR "_move_pallete_temp3";
END_REGION

REGION Network 86
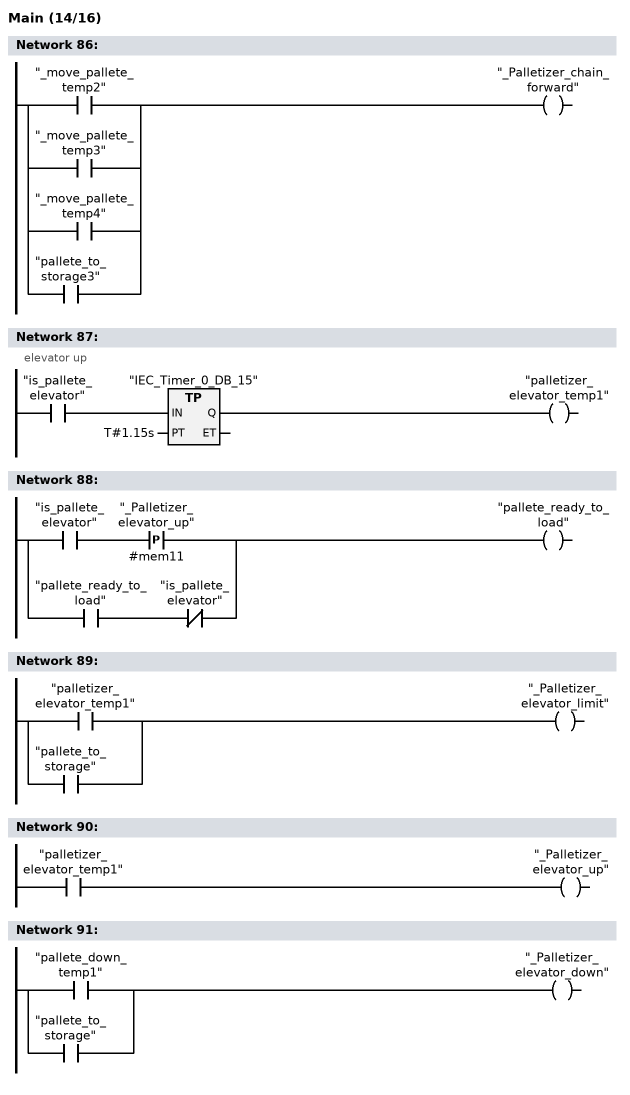
   RUNG wire#powerrail
      Contact( "_move_pallete_temp2" )
      wire#w1
      Coil( "_Palletizer_chain_forward" )
   END_RUNG
   RUNG wire#powerrail
      Contact( "_move_pallete_temp3" )
   END_RUNG wire#w1
   RUNG wire#powerrail
      Contact( "_move_pallete_temp4" )
   END_RUNG wire#w1
   RUNG wire#powerrail
      Contact( "pallete_to_storage3" )
   END_RUNG wire#w1
   // the same network as SCL:
   "_Palletizer_chain_forward" := "_move_pallete_temp2" OR "_move_pallete_temp3" OR "_move_pallete_temp4" OR "pallete_to_storage3";
END_REGION

REGION Network 87
   // elevator up
   "IEC_Timer_0_DB_15".TP(IN := "is_pallete_elevator", PT := T#1.15s);
   "palletizer_elevator_temp1" := "IEC_Timer_0_DB_15".Q;
END_REGION

REGION Network 88
   RUNG wire#powerrail
      Contact( "is_pallete_elevator" )
      P_Contact(operand := "_Palletizer_elevator_up", bit := #mem11)
      wire#w1
      Coil( "pallete_ready_to_load" )
   END_RUNG
   RUNG wire#powerrail
      Contact( "pallete_ready_to_load" )
      I_Contact( "is_pallete_elevator" )
   END_RUNG wire#w1
   // the same network as SCL:
   #_w1 := "is_pallete_elevator" AND "_Palletizer_elevator_up" AND NOT #mem11;   // rising edge of "_Palletizer_elevator_up"
   #mem11 := "_Palletizer_elevator_up";
   "pallete_ready_to_load" := #_w1 OR ("pallete_ready_to_load" AND NOT "is_pallete_elevator");
END_REGION

REGION Network 89
   RUNG wire#powerrail
      Contact( "palletizer_elevator_temp1" )
      wire#w1
      Coil( "_Palletizer_elevator_limit" )
   END_RUNG
   RUNG wire#powerrail
      Contact( "pallete_to_storage" )
   END_RUNG wire#w1
   // the same network as SCL:
   "_Palletizer_elevator_limit" := "palletizer_elevator_temp1" OR "pallete_to_storage";
END_REGION

REGION Network 90
   RUNG wire#powerrail
      Contact( "palletizer_elevator_temp1" )
      Coil( "_Palletizer_elevator_up" )
   END_RUNG
   // the same network as SCL:
   "_Palletizer_elevator_up" := "palletizer_elevator_temp1";
END_REGION

REGION Network 91
   RUNG wire#powerrail
      Contact( "pallete_down_temp1" )
      wire#w1
      Coil( "_Palletizer_elevator_down" )
   END_RUNG
   RUNG wire#powerrail
      Contact( "pallete_to_storage" )
   END_RUNG wire#w1
   // the same network as SCL:
   "_Palletizer_elevator_down" := "pallete_down_temp1" OR "pallete_to_storage";
END_REGION

REGION Network 93: Outputs
   // Set global outputs
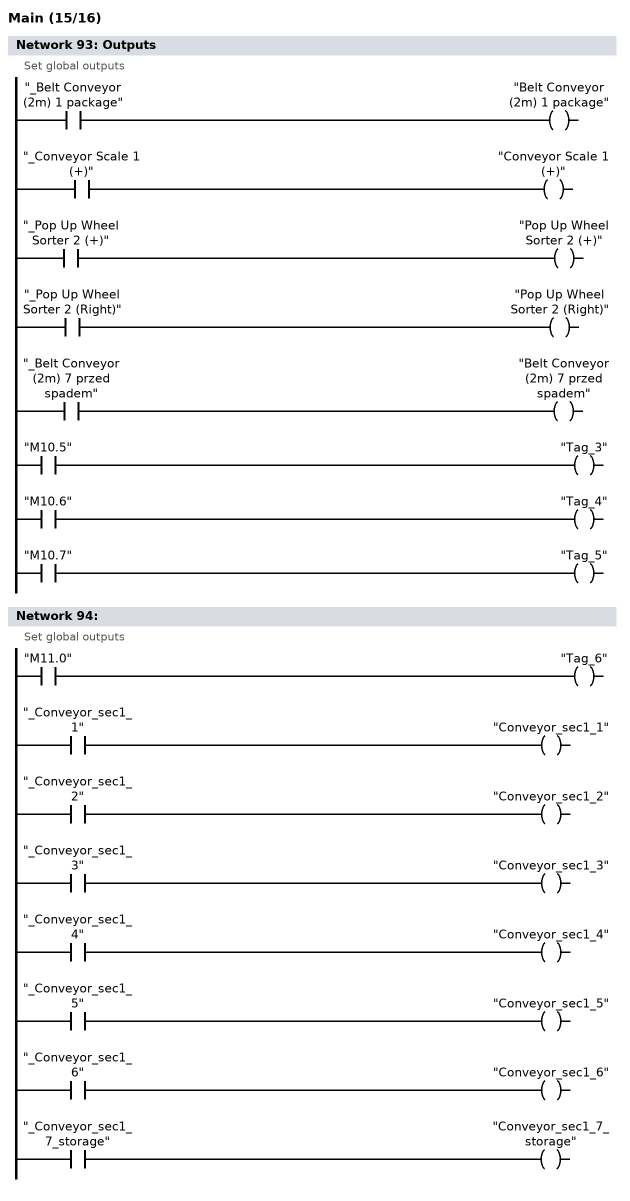
   RUNG wire#powerrail
      Contact( "_Belt Conveyor (2m) 1 package" )
      Coil( "Belt Conveyor (2m) 1 package" )
   END_RUNG
   RUNG wire#powerrail
      Contact( "_Conveyor Scale 1 (+)" )
      Coil( "Conveyor Scale 1 (+)" )
   END_RUNG
   RUNG wire#powerrail
      Contact( "_Pop Up Wheel Sorter 2 (+)" )
      Coil( "Pop Up Wheel Sorter 2 (+)" )
   END_RUNG
   RUNG wire#powerrail
      Contact( "_Pop Up Wheel Sorter 2 (Right)" )
      Coil( "Pop Up Wheel Sorter 2 (Right)" )
   END_RUNG
   RUNG wire#powerrail
      Contact( "_Belt Conveyor (2m) 7 przed spadem" )
      Coil( "Belt Conveyor (2m) 7 przed spadem" )
   END_RUNG
   RUNG wire#powerrail
      Contact( "M10.5" )
      Coil( "Tag_3" )
   END_RUNG
   RUNG wire#powerrail
      Contact( "M10.6" )
      Coil( "Tag_4" )
   END_RUNG
   RUNG wire#powerrail
      Contact( "M10.7" )
      Coil( "Tag_5" )
   END_RUNG
   // the same network as SCL:
   "Belt Conveyor (2m) 1 package" := "_Belt Conveyor (2m) 1 package";
   "Conveyor Scale 1 (+)" := "_Conveyor Scale 1 (+)";
   "Pop Up Wheel Sorter 2 (+)" := "_Pop Up Wheel Sorter 2 (+)";
   "Pop Up Wheel Sorter 2 (Right)" := "_Pop Up Wheel Sorter 2 (Right)";
   "Belt Conveyor (2m) 7 przed spadem" := "_Belt Conveyor (2m) 7 przed spadem";
   "Tag_3" := "M10.5";
   "Tag_4" := "M10.6";
   "Tag_5" := "M10.7";
END_REGION

REGION Network 94
   // Set global outputs
   RUNG wire#powerrail
      Contact( "M11.0" )
      Coil( "Tag_6" )
   END_RUNG
   RUNG wire#powerrail
      Contact( "_Conveyor_sec1_1" )
      Coil( "Conveyor_sec1_1" )
   END_RUNG
   RUNG wire#powerrail
      Contact( "_Conveyor_sec1_2" )
      Coil( "Conveyor_sec1_2" )
   END_RUNG
   RUNG wire#powerrail
      Contact( "_Conveyor_sec1_3" )
      Coil( "Conveyor_sec1_3" )
   END_RUNG
   RUNG wire#powerrail
      Contact( "_Conveyor_sec1_4" )
      Coil( "Conveyor_sec1_4" )
   END_RUNG
   RUNG wire#powerrail
      Contact( "_Conveyor_sec1_5" )
      Coil( "Conveyor_sec1_5" )
   END_RUNG
   RUNG wire#powerrail
      Contact( "_Conveyor_sec1_6" )
      Coil( "Conveyor_sec1_6" )
   END_RUNG
   RUNG wire#powerrail
      Contact( "_Conveyor_sec1_7_storage" )
      Coil( "Conveyor_sec1_7_storage" )
   END_RUNG
   // the same network as SCL:
   "Tag_6" := "M11.0";
   "Conveyor_sec1_1" := "_Conveyor_sec1_1";
   "Conveyor_sec1_2" := "_Conveyor_sec1_2";
   "Conveyor_sec1_3" := "_Conveyor_sec1_3";
   "Conveyor_sec1_4" := "_Conveyor_sec1_4";
   "Conveyor_sec1_5" := "_Conveyor_sec1_5";
   "Conveyor_sec1_6" := "_Conveyor_sec1_6";
   "Conveyor_sec1_7_storage" := "_Conveyor_sec1_7_storage";
END_REGION

REGION Network 95
   // widlak1
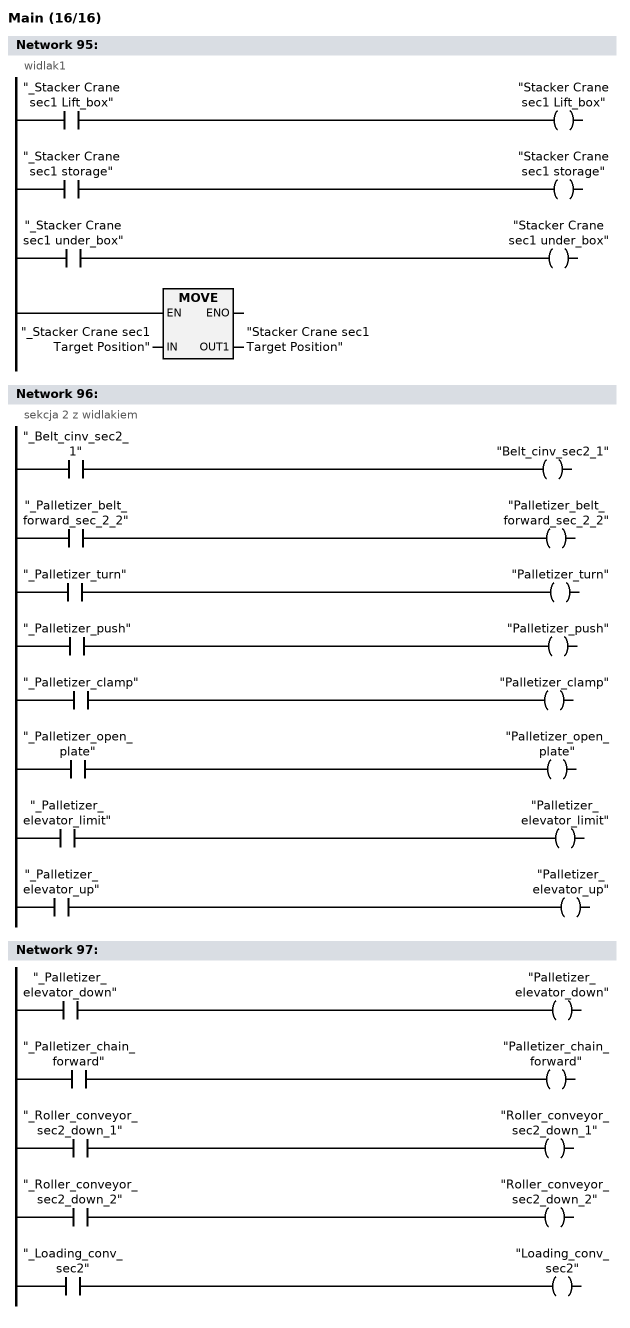
   RUNG wire#powerrail
      Contact( "_Stacker Crane sec1 Lift_box" )
      Coil( "Stacker Crane sec1 Lift_box" )
   END_RUNG
   RUNG wire#powerrail
      Contact( "_Stacker Crane sec1 storage" )
      Coil( "Stacker Crane sec1 storage" )
   END_RUNG
   RUNG wire#powerrail
      Contact( "_Stacker Crane sec1 under_box" )
      Coil( "Stacker Crane sec1 under_box" )
   END_RUNG
   RUNG wire#powerrail
      Move(in := "_Stacker Crane sec1 Target Position", out1 => "Stacker Crane sec1 Target Position")
   END_RUNG
   // the same network as SCL:
   "Stacker Crane sec1 Lift_box" := "_Stacker Crane sec1 Lift_box";
   "Stacker Crane sec1 storage" := "_Stacker Crane sec1 storage";
   "Stacker Crane sec1 under_box" := "_Stacker Crane sec1 under_box";
   "Stacker Crane sec1 Target Position" := "_Stacker Crane sec1 Target Position";
END_REGION

REGION Network 96
   // sekcja 2 z widlakiem
   RUNG wire#powerrail
      Contact( "_Belt_cinv_sec2_1" )
      Coil( "Belt_cinv_sec2_1" )
   END_RUNG
   RUNG wire#powerrail
      Contact( "_Palletizer_belt_forward_sec_2_2" )
      Coil( "Palletizer_belt_forward_sec_2_2" )
   END_RUNG
   RUNG wire#powerrail
      Contact( "_Palletizer_turn" )
      Coil( "Palletizer_turn" )
   END_RUNG
   RUNG wire#powerrail
      Contact( "_Palletizer_push" )
      Coil( "Palletizer_push" )
   END_RUNG
   RUNG wire#powerrail
      Contact( "_Palletizer_clamp" )
      Coil( "Palletizer_clamp" )
   END_RUNG
   RUNG wire#powerrail
      Contact( "_Palletizer_open_plate" )
      Coil( "Palletizer_open_plate" )
   END_RUNG
   RUNG wire#powerrail
      Contact( "_Palletizer_elevator_limit" )
      Coil( "Palletizer_elevator_limit" )
   END_RUNG
   RUNG wire#powerrail
      Contact( "_Palletizer_elevator_up" )
      Coil( "Palletizer_elevator_up" )
   END_RUNG
   // the same network as SCL:
   "Belt_cinv_sec2_1" := "_Belt_cinv_sec2_1";
   "Palletizer_belt_forward_sec_2_2" := "_Palletizer_belt_forward_sec_2_2";
   "Palletizer_turn" := "_Palletizer_turn";
   "Palletizer_push" := "_Palletizer_push";
   "Palletizer_clamp" := "_Palletizer_clamp";
   "Palletizer_open_plate" := "_Palletizer_open_plate";
   "Palletizer_elevator_limit" := "_Palletizer_elevator_limit";
   "Palletizer_elevator_up" := "_Palletizer_elevator_up";
END_REGION

REGION Network 97
   RUNG wire#powerrail
      Contact( "_Palletizer_elevator_down" )
      Coil( "Palletizer_elevator_down" )
   END_RUNG
   RUNG wire#powerrail
      Contact( "_Palletizer_chain_forward" )
      Coil( "Palletizer_chain_forward" )
   END_RUNG
   RUNG wire#powerrail
      Contact( "_Roller_conveyor_sec2_down_1" )
      Coil( "Roller_conveyor_sec2_down_1" )
   END_RUNG
   RUNG wire#powerrail
      Contact( "_Roller_conveyor_sec2_down_2" )
      Coil( "Roller_conveyor_sec2_down_2" )
   END_RUNG
   RUNG wire#powerrail
      Contact( "_Loading_conv_sec2" )
      Coil( "Loading_conv_sec2" )
   END_RUNG
   // the same network as SCL:
   "Palletizer_elevator_down" := "_Palletizer_elevator_down";
   "Palletizer_chain_forward" := "_Palletizer_chain_forward";
   "Roller_conveyor_sec2_down_1" := "_Roller_conveyor_sec2_down_1";
   "Roller_conveyor_sec2_down_2" := "_Roller_conveyor_sec2_down_2";
   "Loading_conv_sec2" := "_Loading_conv_sec2";
END_REGION
END_ORGANIZATION_BLOCK

ORGANIZATION_BLOCK "Startup"   // OB100, LAD, Startup
TITLE = "Complete Restart"
{ S7_Optimized_Access := 'TRUE' }
VERSION : 0.1
   VAR_INPUT
      LostRetentive : Bool;   // True if retentive data are lost
      LostRTC : Bool;   // True if date and time are lost
   END_VAR
BEGIN

REGION Network 1
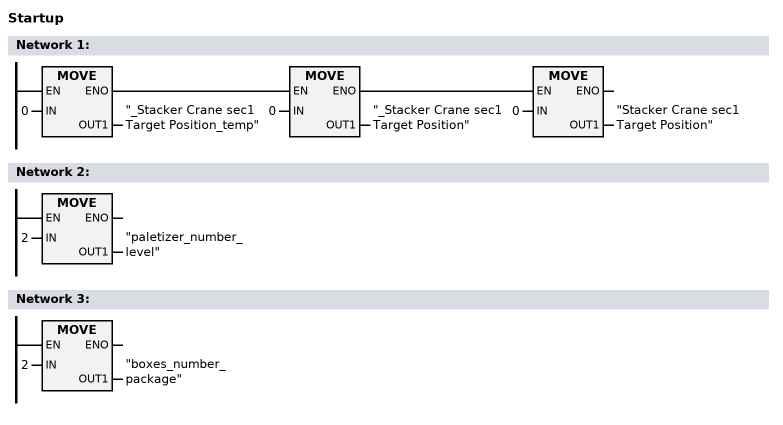
   RUNG wire#powerrail
      Move(in := 0, out1 => "_Stacker Crane sec1 Target Position_temp")
      Move(in := 0, out1 => "_Stacker Crane sec1 Target Position")
      Move(in := 0, out1 => "Stacker Crane sec1 Target Position")
   END_RUNG
   // the same network as SCL:
   "_Stacker Crane sec1 Target Position_temp" := 0;
   "_Stacker Crane sec1 Target Position" := 0;
   "Stacker Crane sec1 Target Position" := 0;
END_REGION

REGION Network 2
   RUNG wire#powerrail
      Move(in := 2, out1 => "paletizer_number_level")
   END_RUNG
   // the same network as SCL:
   "paletizer_number_level" := 2;
END_REGION

REGION Network 3
   RUNG wire#powerrail
      Move(in := 2, out1 => "boxes_number_package")
   END_RUNG
   // the same network as SCL:
   "boxes_number_package" := 2;
END_REGION
END_ORGANIZATION_BLOCK

(* ===== HMI "HMI_RT_1" =====
system functions are stored by id; their names below are inferred from use
connection "HMI_Connection_1": ETHERNET, S7_1200_OMS

HMI tags "Default tag table"
   "paletizer_counter" : Int = PLC paletizer_counter AT %MW6, 1 s
   "boxes_counter" : Int = PLC boxes_counter AT %MW8, 1 s
   "paletizer_number_level" : Int = PLC paletizer_number_level AT %MW16, 1 s
   "boxes_number_package" : Int = PLC boxes_number_package AT %MW18, 1 s

Template "Template_1" 800x480
   Button "Exit" at 720,420 size 78x58; TextOff 'Exit'; PictureOff "ExitRuntime_TP900_Comfort_TR"; PictureOn "ExitRuntime_TP900_Comfort_TR"
      on Release: StopRuntime(0)
   Button "Template_Button" at 640,420 size 78x58; TextOff 'Text'
   Button "Template_Button_1" at 560,420 size 78x58; TextOff 'Text'
   Button "Template_Button_2" at 480,420 size 78x58; TextOff 'Text'
   Button "Template_Button_3" at 400,420 size 78x58; TextOff 'Text'
   Button "Template_Button_4" at 321,420 size 78x58; TextOff 'Text'
   Button "Template_Button_5" at 241,420 size 78x58; TextOff 'Text'
   Button "Template_Button_6" at 161,420 size 78x58; TextOff 'Text'
   Button "Alarms" at 81,420 size 78x58; TextOff 'Alarms'; PictureOff "AlarmDisplay_TP900_Comfort_TR"; PictureOn "AlarmDisplay_TP900_Comfort_TR"
      on Release: function_ef3f5d25("Alarm window_Unacknowledged", -1)
   Button "Start screen" at 1,420 size 78x58; TextOff 'Start screen'; PictureOff "NavigateHome_TP900_Comfort_TR"; PictureOn "NavigateHome_TP900_Comfort_TR"
      on Release: ActivateScreen("Root screen", 0)

screen "Root screen" 800x480, template "Template_1"
   IOField "I/O field_1" at 579,74 size 96x32; FormatPattern 999
      ProcessValue <- "paletizer_counter"
   IOField "I/O field_2" at 579,216 size 96x32; FormatPattern 999
      ProcessValue <- "boxes_counter"
   IOField "I/O field_3" at 60,76 size 96x32; FormatPattern 9
      ProcessValue <- "paletizer_number_level"
   TextField "Text field_1" at 64,37 size 92x20; Text 'Ile warstw?'
   TextField "Text field_2" at 551,181 size 159x20; Text 'Załadowane skrzynki'
   TextField "Text field_3" at 566,37 size 114x20; Text 'Ułożone paczki'
   IOField "I/O field_4" at 63,216 size 96x32; FormatPattern 9
      ProcessValue <- "boxes_number_package"
   TextField "Text field_4" at 71,181 size 88x20; Text 'Ile paczek?'
*)